(* CODESYS project boiler_olgovo_22_10_2019.project
   Company: syat
   Title: boiler_olgovo
   Author: User
   Version: 0.0.0.207

Project tree, tasks and I/O mapping:
  MyController : TM241CE40T/U, Schneider Electric, order no. TM241CE40T/U, version 4.0.6.18
      settings: OPCUA enable = False
    application Application
      libraries: CAA Real Time Clock Extern, 3.5.1.0 (CAA Technical Workgroup); SysTimeRtc, 3.5.1.0 (System)
      task MAST (cyclic, interval 20 ms, priority 15, watchdog 100 ms x 1) calls analog_input, IN_A1_A12_A14_A17, MB_IN, get_data_from_CKM, reset_flowmetr, send_data_to_flowmeter, zadanie_for_m1_m2, get_data_from_flowmetr, BURNERS_GAZ_GRU, avg, day_mode, HVO_HEATER, connection, DYMOHODS, RECIRCULATIONS_M5_M6_M7, POUWER_BOILER, ALL_ERR, zadanie_for_burner, set_time, ERR_SENSER, SECURITY_BOILER, VALVE_FEEDER_PUMP_FEEDERS_M3_M4, NET_PUMPS_M1_M2, TRHD_PEREPUSK, ZATVORS, MB_OUT, OUT_PIN, send_data_to_flowmeter
      global variables GVL
      program OUT_PIN [ST]
      program IN_A1_A12_A14_A17 [ST]
      FB/
        function block VALVE_FEEDER [LD]
        function block PUMP [LD]
        function block VALVE [LD]
        function block BURNER_SMALL [LD]
        function send_to_ckm [LD]
        function block VALVE_TRHD [LD]
        function block PUMP_PCH [LD]
        function block VALVE_DYMOHOD [LD]
        function block VALVE_TRHD_PEREPUSK [LD]
        function block BURNER_BIG [LD]
      program MB_OUT [ST]
      program MB_IN [ST]
      program DYMOHODS [LD]
      program ZATVORS [LD]
      program TRHD_PEREPUSK [LD]
      program HVO_HEATER [LD]
      program RECIRCULATIONS_M5_M6_M7 [LD]
      program NET_PUMPS_M1_M2 [LD]
      program VALVE_FEEDER_PUMP_FEEDERS_M3_M4 [LD]
      program SECURITY_BOILER [LD]
      program BURNERS_GAZ_GRU [LD]
      program POUWER_BOILER [ST]
      program get_data_from_flowmetr [ST]
      program get_data_from_CKM [ST]
      program get_data_from_gaz_korr [LD]
      program zadanie_for_burner [ST]
      program ERR_SENSER [LD]
      program ALL_ERR [LD]
      global variables GVL_RETAIN
      A_TESTS/
        program zadanie_for_m1_m2 [ST]
        program zadanie_for_pch_m7 [ST]
        program zadanie_m7 [FBD]
        program zadanie_m1_m2 [FBD]
      RecipeManager
      global variables GVL_state_valve
      global variables GVL_STATE_PUMP
      global variables GVL_grafik
      program send_data_to_flowmeter [LD]
      program reset_flowmetr [ST]
      program set_time [CFC]
      program day_mode [CFC]
      program analog_input [LD]
      program avg [CFC]
      program connection [LD]
    DI : Digital Inputs, Schneider Electric, version 4.0.6.18
        input  idwDI_IDW0 : DWORD  // IDW0
        input  X0 : BOOL  // IDW0.I0
        input  X1 : BOOL  // IDW0.I1
        input  X2 : BOOL  // IDW0.I2
        input  X3 : BOOL  // IDW0.I3
        input  X4 : BOOL  // IDW0.I4
        input  X5 : BOOL  // IDW0.I5
        input  X6 : BOOL  // IDW0.I6
        input  X7 : BOOL  // IDW0.I7
        input  X8 : BOOL  // IDW0.I8
        input  X9 : BOOL  // IDW0.I9
        input  X10 : BOOL  // IDW0.I10
        input  X11 : BOOL  // IDW0.I11
        input  X12 : BOOL  // IDW0.I12
        input  X13 : BOOL  // IDW0.I13
        input  X14 : BOOL  // IDW0.I14
        input  X15 : BOOL  // IDW0.I15
        input  X16 : BOOL  // IDW0.I16
        input  X17 : BOOL  // IDW0.I17
        input  X18 : BOOL  // IDW0.I18
        input  X19 : BOOL  // IDW0.I19
        input  X20 : BOOL  // IDW0.I20
        input  X21 : BOOL  // IDW0.I21
        input  X22 : BOOL  // IDW0.I22
        input  X23 : BOOL  // IDW0.I23
        input  ibDI_IB1 : BYTE  // IB1
    DQ : Digital Outputs, Schneider Electric, version 4.0.6.18
        output Y0 : BOOL  // QW0.Q0
        output Y1 : BOOL  // QW0.Q1
        output Y2 : BOOL  // QW0.Q2
        output Y3 : BOOL  // QW0.Q3
        output Y4 : BOOL  // QW0.Q4
        output Y5 : BOOL  // QW0.Q5
        output Y6 : BOOL  // QW0.Q6
        output Y7 : BOOL  // QW0.Q7
        output Y8 : BOOL  // QW0.Q8
        output Y9 : BOOL  // QW0.Q9
        output Y10 : BOOL  // QW0.Q10
        output Y11 : BOOL  // QW0.Q11
        output Y12 : BOOL  // QW0.Q12
        output Y13 : BOOL  // QW0.Q13
        output Y14 : BOOL  // QW0.Q14
        output Y15 : BOOL  // QW0.Q15
        output qbDQ_QB1 : BYTE  // QB1
        unmapped channels: QW0
    Counters : Counters, Schneider Electric, version 4.0.6.18
    Pulse_Generators : Pulse Generators, Schneider Electric, version 4.0.6.18
    Cartridge_1 : Cartridge, Schneider Electric, version 4.0.6.18
    Cartridge_2 : Cartridge, Schneider Electric, version 4.0.6.18
    IO_Bus : IO bus - TM3, Schneider Electric, version 4.0.6.18
      A1_7 : TM3TI4/G, Schneider Electric, order no. TM3TI4/G, version 1.0.1.5
          settings: KPI Configuration.KPI Configuration[0] = 35; KPI Configuration.KPI Configuration[1] = 35; KPI Configuration.KPI Configuration[2] = 35; KPI Configuration.KPI Configuration[3] = 35; KPI Configuration.KPI Configuration[5] = 0; KPI Configuration.KPI Configuration[7] = 0; KPI Configuration.KPI Configuration[9] = 0; KPI Configuration.KPI Configuration[11] = 0; KPI Configuration.KPI Configuration[12] = 32; KPI Configuration.KPI Configuration[13] = 78; KPI Configuration.KPI Configuration[14] = 32; KPI Configuration.KPI Configuration[15] = 78; KPI Configuration.KPI Configuration[16] = 32; KPI Configuration.KPI Configuration[17] = 78; KPI Configuration.KPI Configuration[18] = 32; KPI Configuration.KPI Configuration[19] = 78; KPI Configuration.KPI Configuration[20] = 10; KPI Configuration.KPI Configuration[22] = 10; KPI Configuration.KPI Configuration[24] = 10; KPI Configuration.KPI Configuration[26] = 10
          input  PT9 : INT  // IW0
          input  PT10 : INT  // IW1
          input  PT11 : INT  // IW2
          input  PT01 : INT  // IW3
          input  ERR_PT9 : BYTE  // IBStatusIW0
          input  ERR_PT10 : BYTE  // IBStatusIW1
          input  ERR_PT11 : BYTE  // IBStatusIW2
          input  ERR_PT01 : BYTE  // IBStatusIW3
      A1_6 : TM3AI8/G, Schneider Electric, order no. TM3AI8/G, version 1.0.0.17
          settings: KPI Configuration.KPI Configuration[0] = 35; KPI Configuration.KPI Configuration[1] = 35; KPI Configuration.KPI Configuration[2] = 35; KPI Configuration.KPI Configuration[3] = 35; KPI Configuration.KPI Configuration[4] = 35; KPI Configuration.KPI Configuration[5] = 35; KPI Configuration.KPI Configuration[6] = 35; KPI Configuration.KPI Configuration[7] = 35; KPI Configuration.KPI Configuration[9] = 0; KPI Configuration.KPI Configuration[11] = 0; KPI Configuration.KPI Configuration[13] = 0; KPI Configuration.KPI Configuration[15] = 0; KPI Configuration.KPI Configuration[17] = 0; KPI Configuration.KPI Configuration[19] = 0; KPI Configuration.KPI Configuration[21] = 0; KPI Configuration.KPI Configuration[23] = 0; KPI Configuration.KPI Configuration[24] = 32; KPI Configuration.KPI Configuration[25] = 78; KPI Configuration.KPI Configuration[26] = 32; KPI Configuration.KPI Configuration[27] = 78; KPI Configuration.KPI Configuration[28] = 32; KPI Configuration.KPI Configuration[29] = 78; KPI Configuration.KPI Configuration[30] = 32; KPI Configuration.KPI Configuration[31] = 78; KPI Configuration.KPI Configuration[32] = 32; KPI Configuration.KPI Configuration[33] = 78; KPI Configuration.KPI Configuration[34] = 32; KPI Configuration.KPI Configuration[35] = 78; KPI Configuration.KPI Configuration[36] = 32; KPI Configuration.KPI Configuration[37] = 78; KPI Configuration.KPI Configuration[38] = 32; KPI Configuration.KPI Configuration[39] = 78; KPI Configuration.KPI Configuration[40] = 10; KPI Configuration.KPI Configuration[42] = 10; KPI Configuration.KPI Configuration[44] = 10; KPI Configuration.KPI Configuration[46] = 10; KPI Configuration.KPI Configuration[48] = 10; KPI Configuration.KPI Configuration[50] = 10; KPI Configuration.KPI Configuration[52] = 10; KPI Configuration.KPI Configuration[54] = 10
          input  PT1 : INT  // IW0
          input  PT2 : INT  // IW1
          input  PT3 : INT  // IW2
          input  PT4 : INT  // IW3
          input  PT5 : INT  // IW4
          input  PT6 : INT  // IW5
          input  PT7 : INT  // IW6
          input  PT8 : INT  // IW7
          input  ERR_PT1 : BYTE  // IBStatusIW0
          input  ERR_PT2 : BYTE  // IBStatusIW1
          input  ERR_PT3 : BYTE  // IBStatusIW2
          input  ERR_PT4 : BYTE  // IBStatusIW3
          input  ERR_PT5 : BYTE  // IBStatusIW4
          input  ERR_PT6 : BYTE  // IBStatusIW5
          input  ERR_PT7 : BYTE  // IBStatusIW6
          input  ERR_PT8 : BYTE  // IBStatusIW7
      A1_5 : TM3AI8/G, Schneider Electric, order no. TM3AI8/G, version 1.0.0.17
          settings: KPI Configuration.KPI Configuration[0] = 35; KPI Configuration.KPI Configuration[1] = 35; KPI Configuration.KPI Configuration[2] = 35; KPI Configuration.KPI Configuration[3] = 35; KPI Configuration.KPI Configuration[4] = 35; KPI Configuration.KPI Configuration[5] = 35; KPI Configuration.KPI Configuration[6] = 35; KPI Configuration.KPI Configuration[7] = 35; KPI Configuration.KPI Configuration[9] = 0; KPI Configuration.KPI Configuration[11] = 0; KPI Configuration.KPI Configuration[13] = 0; KPI Configuration.KPI Configuration[15] = 0; KPI Configuration.KPI Configuration[17] = 0; KPI Configuration.KPI Configuration[19] = 0; KPI Configuration.KPI Configuration[21] = 0; KPI Configuration.KPI Configuration[23] = 0; KPI Configuration.KPI Configuration[24] = 32; KPI Configuration.KPI Configuration[25] = 78; KPI Configuration.KPI Configuration[26] = 32; KPI Configuration.KPI Configuration[27] = 78; KPI Configuration.KPI Configuration[28] = 32; KPI Configuration.KPI Configuration[29] = 78; KPI Configuration.KPI Configuration[30] = 32; KPI Configuration.KPI Configuration[31] = 78; KPI Configuration.KPI Configuration[32] = 32; KPI Configuration.KPI Configuration[33] = 78; KPI Configuration.KPI Configuration[34] = 208; KPI Configuration.KPI Configuration[35] = 7; KPI Configuration.KPI Configuration[36] = 32; KPI Configuration.KPI Configuration[37] = 78; KPI Configuration.KPI Configuration[38] = 32; KPI Configuration.KPI Configuration[39] = 78; KPI Configuration.KPI Configuration[40] = 10; KPI Configuration.KPI Configuration[42] = 10; KPI Configuration.KPI Configuration[44] = 10; KPI Configuration.KPI Configuration[46] = 10; KPI Configuration.KPI Configuration[48] = 10; KPI Configuration.KPI Configuration[50] = 10; KPI Configuration.KPI Configuration[52] = 10; KPI Configuration.KPI Configuration[54] = 10;
            KPI Configuration.KPI Configuration[61] = 1; KPI Configuration.KPI Configuration[62] = 1
          input  TT9 : INT  // IW0
          input  TT10 : INT  // IW1
          input  TT11 : INT  // IW2
          input  TT12 : INT  // IW3
          input  TT13 : INT  // IW4
          input  TT14 : INT  // IW5
          input  TT15 : INT  // IW6
          input  TT16 : INT  // IW7
          input  ERR_TT9 : BYTE  // IBStatusIW0
          input  ERR_TT10 : BYTE  // IBStatusIW1
          input  ERR_TT11 : BYTE  // IBStatusIW2
          input  ERR_TT12 : BYTE  // IBStatusIW3
          input  ERR_TT13 : BYTE  // IBStatusIW4
          input  ERR_TT14 : BYTE  // IBStatusIW5
          input  ERR_TT15 : BYTE  // IBStatusIW6
          input  ERR_TT16 : BYTE  // IBStatusIW7
      A1_4 : TM3AI8/G, Schneider Electric, order no. TM3AI8/G, version 1.0.0.17
          settings: KPI Configuration.KPI Configuration[0] = 35; KPI Configuration.KPI Configuration[1] = 35; KPI Configuration.KPI Configuration[2] = 35; KPI Configuration.KPI Configuration[3] = 35; KPI Configuration.KPI Configuration[4] = 35; KPI Configuration.KPI Configuration[5] = 35; KPI Configuration.KPI Configuration[6] = 35; KPI Configuration.KPI Configuration[7] = 35; KPI Configuration.KPI Configuration[9] = 0; KPI Configuration.KPI Configuration[11] = 0; KPI Configuration.KPI Configuration[13] = 0; KPI Configuration.KPI Configuration[15] = 0; KPI Configuration.KPI Configuration[17] = 0; KPI Configuration.KPI Configuration[19] = 0; KPI Configuration.KPI Configuration[21] = 0; KPI Configuration.KPI Configuration[23] = 0; KPI Configuration.KPI Configuration[24] = 32; KPI Configuration.KPI Configuration[25] = 78; KPI Configuration.KPI Configuration[26] = 32; KPI Configuration.KPI Configuration[27] = 78; KPI Configuration.KPI Configuration[28] = 32; KPI Configuration.KPI Configuration[29] = 78; KPI Configuration.KPI Configuration[30] = 32; KPI Configuration.KPI Configuration[31] = 78; KPI Configuration.KPI Configuration[32] = 32; KPI Configuration.KPI Configuration[33] = 78; KPI Configuration.KPI Configuration[34] = 32; KPI Configuration.KPI Configuration[35] = 78; KPI Configuration.KPI Configuration[36] = 32; KPI Configuration.KPI Configuration[37] = 78; KPI Configuration.KPI Configuration[38] = 32; KPI Configuration.KPI Configuration[39] = 78; KPI Configuration.KPI Configuration[40] = 10; KPI Configuration.KPI Configuration[42] = 10; KPI Configuration.KPI Configuration[44] = 10; KPI Configuration.KPI Configuration[46] = 10; KPI Configuration.KPI Configuration[48] = 10; KPI Configuration.KPI Configuration[50] = 10; KPI Configuration.KPI Configuration[52] = 10; KPI Configuration.KPI Configuration[54] = 10
          input  TT1 : INT  // IW0
          input  TT2 : INT  // IW1
          input  TT3 : INT  // IW2
          input  TT4 : INT  // IW3
          input  TT5 : INT  // IW4
          input  TT6 : INT  // IW5
          input  TT7 : INT  // IW6
          input  TT8 : INT  // IW7
          input  ERR_TT1 : BYTE  // IBStatusIW0
          input  ERR_TT2 : BYTE  // IBStatusIW1
          input  ERR_TT3 : BYTE  // IBStatusIW2
          input  ERR_TT4 : BYTE  // IBStatusIW3
          input  ERR_TT5 : BYTE  // IBStatusIW4
          input  ERR_TT6 : BYTE  // IBStatusIW5
          input  ERR_TT7 : BYTE  // IBStatusIW6
          input  ERR_TT8 : BYTE  // IBStatusIW7
      A1_3 : TM3DQ32TK, Schneider Electric, order no. TM3DQ32TK, version 1.0.1.3
          output IY0 : BOOL  // QD0.Q0
          output IY1 : BOOL  // QD0.Q1
          output IY2 : BOOL  // QD0.Q2
          output IY3 : BOOL  // QD0.Q3
          output IY4 : BOOL  // QD0.Q4
          output IY5 : BOOL  // QD0.Q5
          output IY6 : BOOL  // QD0.Q6
          output IY7 : BOOL  // QD0.Q7
          output IY8 : BOOL  // QD0.Q8
          output IY9 : BOOL  // QD0.Q9
          output IY10 : BOOL  // QD0.Q10
          output IY11 : BOOL  // QD0.Q11
          output IY12 : BOOL  // QD0.Q12
          output IY13 : BOOL  // QD0.Q13
          output IY14 : BOOL  // QD0.Q14
          output IY15 : BOOL  // QD0.Q15
          output IY16 : BOOL  // QD0.Q16
          output IY17 : BOOL  // QD0.Q17
          output IY18 : BOOL  // QD0.Q18
          output IY19 : BOOL  // QD0.Q19
          output IY20 : BOOL  // QD0.Q20
          output IY25 : BOOL  // QD0.Q25
          unmapped channels: QD0
      A1_1 : TM3DI32K, Schneider Electric, order no. TM3DI32K, version 1.0.1.3
          input  idwA1_1_ID0 : DWORD  // ID0
          input  IX0 : BOOL  // ID0.I0
          input  IX1 : BOOL  // ID0.I1
          input  IX2 : BOOL  // ID0.I2
          input  IX3 : BOOL  // ID0.I3
          input  IX4 : BOOL  // ID0.I4
          input  IX5 : BOOL  // ID0.I5
          input  IX6 : BOOL  // ID0.I6
          input  IX7 : BOOL  // ID0.I7
          input  IX8 : BOOL  // ID0.I8
          input  IX9 : BOOL  // ID0.I9
          input  IX10 : BOOL  // ID0.I10
          input  IX11 : BOOL  // ID0.I11
          input  IX12 : BOOL  // ID0.I12
          input  IX13 : BOOL  // ID0.I13
          input  IX14 : BOOL  // ID0.I14
          input  IX15 : BOOL  // ID0.I15
          input  IX16 : BOOL  // ID0.I16
          input  IX17 : BOOL  // ID0.I17
          input  IX18 : BOOL  // ID0.I18
          input  IX19 : BOOL  // ID0.I19
          input  IX20 : BOOL  // ID0.I20
          input  IX21 : BOOL  // ID0.I21
          input  IX22 : BOOL  // ID0.I22
          input  IX23 : BOOL  // ID0.I23
          input  IX24 : BOOL  // ID0.I24
          input  IX25 : BOOL  // ID0.I25
          input  IX26 : BOOL  // ID0.I26
          input  IX27 : BOOL  // ID0.I27
          input  IX28 : BOOL  // ID0.I28
          input  IX29 : BOOL  // ID0.I29
          input  IX30 : BOOL  // ID0.I30
          input  IX31 : BOOL  // ID0.I31
      A1_2 : TM3DI32K, Schneider Electric, order no. TM3DI32K, version 1.0.1.3
          input  IIX0 : BOOL  // ID0.I0
          input  IIX1 : BOOL  // ID0.I1
          input  IIX6 : BOOL  // ID0.I6
          input  IIX7 : BOOL  // ID0.I7
          input  IIX12 : BOOL  // ID0.I12
          input  IIX15 : BOOL  // ID0.I15
          unmapped channels: ID0
    COM_Bus : COM bus, Schneider Electric, version 4.0.6.18
    Ethernet_1 : Ethernet Network, Schneider Electric, version 4.0.6.18
        settings: IPAddress = [192, 168, 0, 32]; SubnetMask = [255, 255, 255, 0]; GatewayAddress = [192, 168, 0, 30]; DeviceName = 'plc_olgovo'; WebServer = TRUE; FTP Server = TRUE; SoMachine Protocol = TRUE; Modbus Server = TRUE; NetManage Protocol = TRUE; SNMP protocol = TRUE; Enable Routing = FALSE; WebVisu protocol = TRUE; DHCP Server Active = TRUE
    Serial_Line_1 : Serial line, Schneider Electric, version 4.0.6.18
      ASCII_Manager : ASCII Manager, Schneider Electric, version 4.0.0.2
    Serial_Line_2 : Serial line, Schneider Electric, version 4.0.6.18
      Modbus_IOScanner : Modbus IOScanner, Schneider Electric, version 3.5.3.8
          settings: Transmission = 'RTU'; ResponseTimeout = 1000; TimeBetweenFrames = 5
        Generic_Modbus_Slave : Generic Modbus Slave, Schneider Electric, version 3.5.3.9
            settings: SlaveAddress = 9; ResponseTimeout = 1000; Channel 1.Function Code = 4; Channel 1.Read Offset = 16#8000; Channel 1.Read Length = 2; Channel 1.Write Offset = 0; Channel 1.Write Length = 0; Channel 1.Cycle Time = 100; Channel 2.Function Code = 4; Channel 2.Read Offset = 16#C000; Channel 2.Read Length = 76; Channel 2.Write Offset = 0; Channel 2.Write Length = 0; Channel 2.Cycle Time = 100
            input  Application.skm_number_arr : ARRAY[0..1] OF WORD  // Channel 1
            input  Application.skm_all : ARRAY[0..75] OF WORD  // Channel 2
        OVEN : Generic Modbus Slave, Schneider Electric, version 3.5.3.9
            settings: SlaveAddress = 16; ResponseTimeout = 100; Channel 1.Function Code = 3; Channel 1.Read Offset = 16#0001; Channel 1.Read Length = 1; Channel 1.Write Offset = 0; Channel 1.Write Length = 0; Channel 1.Cycle Time = 100; Channel 2.Function Code = 3; Channel 2.Read Offset = 16#0007; Channel 2.Read Length = 1; Channel 2.Write Offset = 0; Channel 2.Write Length = 0; Channel 2.Cycle Time = 100
            input  Application.POSITION_VALVE_PEREPUSK : WORD  // Channel 1.Channel 1[0]
            input  Application.POSITION_VALVE_HEATER : WORD  // Channel 2.Channel 2[0]
            unmapped channels: Channel 1, Channel 2
        OVEN_OUT : Generic Modbus Slave, Schneider Electric, version 3.5.3.9
            settings: SlaveAddress = 17; ResponseTimeout = 101; Channel 1.Function Code = 16; Channel 1.Read Offset = 0; Channel 1.Read Length = 0; Channel 1.Write Offset = 16#0000; Channel 1.Write Length = 1; Channel 1.Cycle Time = 100; Channel 2.Function Code = 16; Channel 2.Read Offset = 0; Channel 2.Read Length = 0; Channel 2.Write Offset = 16#0001; Channel 2.Write Length = 1; Channel 2.Cycle Time = 100; Channel 3.Function Code = 16; Channel 3.Read Offset = 0; Channel 3.Read Length = 0; Channel 3.Write Offset = 16#0002; Channel 3.Write Length = 1; Channel 3.Cycle Time = 100
            output Application.PCH_PUMP_M1_ZADANIE : ARRAY[0..0] OF WORD  // Channel 1
            output Application.PCH_PUMP_M2_ZADANIE : ARRAY[0..0] OF WORD  // Channel 2
            output Application.PCH_PUMP_M7_ZADANIE : ARRAY[0..0] OF WORD  // Channel 3
        ek270a : Generic Modbus Slave, Schneider Electric, version 3.5.3.9
            settings: ek270.Function Code = 3; ek270.Read Offset = 16#0146; ek270.Read Length = 2; ek270.Write Offset = 0; ek270.Write Length = 0; ek270.Cycle Time = 100; Channel 2.Function Code = 3; Channel 2.Read Offset = 16#0148; Channel 2.Read Length = 2; Channel 2.Write Offset = 0; Channel 2.Write Length = 0; Channel 2.Cycle Time = 100; Channel 3.Function Code = 3; Channel 3.Read Offset = 16#0064; Channel 3.Read Length = 2; Channel 3.Write Offset = 0; Channel 3.Write Length = 0; Channel 3.Cycle Time = 100; Channel 4.Function Code = 3; Channel 4.Read Offset = 16#0066; Channel 4.Read Length = 2; Channel 4.Write Offset = 0; Channel 4.Write Length = 0; Channel 4.Cycle Time = 100
            input  Q_s : WORD  // ek270.ek270[0]
            input  Q_l : WORD  // ek270.ek270[1]
            input  Qb_s : WORD  // Channel 2.Channel 2[0]
            input  Qb_l : WORD  // Channel 2.Channel 2[1]
            input  V_s : WORD  // Channel 3.Channel 3[0]
            input  V_l : WORD  // Channel 3.Channel 3[1]
            input  Vb_s : WORD  // Channel 4.Channel 4[0]
            input  Vb_l : WORD  // Channel 4.Channel 4[1]
            unmapped channels: ek270, Channel 2, Channel 3, Channel 4
  FdtConnections : FDT Connections, Schneider Electric, version 1.0.0.2
  A_TESTS/
    program get_data_from_oven [ST]
    program zadanie_for_m1_m2 [ST]
    program zadanie_for_pch_m7 [ST]
    program zadanie_m7 [FBD]
    program zadanie_m1_m2 [FBD]
*)

// MyController/Application/GVL
VAR_GLOBAL
	
start_test : BOOL;

//БЛОК ДЛЯ ОБМЕНА С РАСХОДОМЕРОМ ======НАЧАЛО======	
  	FLOW_BOILER_1 AT %MD500: REAL;
	FLOW_BOILER_2 AT %MD501: REAL;
	fl_g_s AT %MW1004: WORD;
	fl_g_l AT %MW1006: WORD;
	FLOW_GAZ AT %MD502: DWORD;
	V_gaz AT %MD506:DWORD;
	//FLOW_BOILER И FL_BOILER ДОЛЖНЫ ССЫЛАТЬСЯ НА ОДНУ ПАМЯТЬ
	FL_BOILER_1 AT %MD500: DWORD;
	FL_BOILER_2 AT %MD501: DWORD;
	
	RASHOD_WATER AT %MW503: WORD;
	FL_HVO AT %MD504: DWORD;
	
//БЛОК ДЛЯ ОБМЕНА С РАСХОДОМЕРОМ ======КОЕЦ======
	
//БЛОК ДЛЯ ОБМЕНА С ОВЕНОМ ======НАЧАЛО======	
  	step: INT;
	POSITION_VALVE_PEREPUSK: INT;
	POSITION_VALVE_HEATER: INT; 
  	data_to_send: ARRAY[0..10] OF BYTE; 
  	resv_data_from_flowmtr_ADR6: ARRAY[0..10] OF BYTE;
	resv_data_from_flowmtr_ADR7: ARRAY[0..10] OF BYTE;
	resv_data_from_flowmtr_ADR8: ARRAY[0..10] OF BYTE;
	resv_data_from_ckm: ARRAY[0..120] OF BYTE;
	good: BOOL;
//БЛОК ДЛЯ ОБМЕНА С ОВЕНОМ ======КОЕЦ======

//БЛОК ОПИСАНИЯ ВХОДОВ А1_1  A1_2 =============НАЧАЛО=======
	ERR_PCH_PUMP_CYRCULATION AT %MX400.0: BOOL;
	ERR_PUMP1_CYRCULATION AT %MX400.1: BOOL;
	ERR_PUMP2_CYRCULATION AT %MX400.2: BOOL;
	ERR_PCH_PUMP1_NET AT %MX400.3: BOOL;
	ERR_PCH_PUMP2_NET AT %MX400.4: BOOL;
	ERR_M3_FEEDER AT %MX400.5: BOOL;
	ERR_M4_FEEDER AT %MX400.6: BOOL;
	VALVE_GAZ_OPENED AT %MX400.7: BOOL;
	VALVE_GAZ_CLOSED AT %MX400.8: BOOL;
	ERR_DEGAZATOR AT %MX400.9: BOOL;
	FIRE AT %MX400.10: BOOL;
	BREAKE AT %MX400.11: BOOL;
	N0_SECURITY AT %MX400.12: BOOL;
	SECURITY AT %MX400.13: BOOL;
	ERR_GAZ AT %MX400.14: BOOL;
	ERR_BURNER1 AT %MX400.15: BOOL;
	

	BTN_HAND_MODE_PUMPS: BOOL;
	BTN_AUTO_MODE_PUMPS:BOOL;
	BTN_HAND_MODE_BOILERS: BOOL;
	BTN_AUTO_MODE_BOILERS:BOOL;
	BTN_HAND_MODE_VALVES: BOOL;
	BTN_AUTO_MODE_VALVES:BOOL;
	BTN_START_BURNER: BOOL;
//БЛОК ОПИСАНИЯ ВХОДОВ А1_1 A1_2 =============КОНЕЦ========

//БЛОК ОПИСАНИЯ ВХОДОВ А1 =============НАЧАЛО=======
	ERR_BURNER2 AT %MX402.0: BOOL;
	BURNER2_WORKS AT %MX402.1: BOOL;
	DYMOHOD1_OPENED AT %MX402.2: BOOL;
	DYMOHOD1_CLOSED AT %MX402.3: BOOL;
	ZATVOR1_OPENED AT %MX402.4: BOOL;
	ZATVOR1_CLOSED AT %MX402.5: BOOL;
	DYMOHOD2_OPENED AT %MX402.6: BOOL;
	DYMOHOD2_CLOSED AT %MX402.7: BOOL;
	ZATVOR2_OPENED AT %MX402.8: BOOL;
	ZATVOR2_CLOSED AT %MX402.9: BOOL;
	FEEDER_OPENED AT %MX402.10: BOOL;
	FEEDER_CLOSED AT %MX402.11: BOOL;
	HVO_OPENED AT %MX402.12: BOOL;
	HVO_CLOSED AT %MX402.13: BOOL;
	PEREPUSK_OPENED AT %MX402.14: BOOL;
	PEREPUSK_CLOSED AT %MX402.15: BOOL;
		
//БЛОК ОПИСАНИЯ ВХОДОВ А1 =============КОНЕЦ========



//БЛОК ОПИСАНИЯ ВЫХОДОВ А1 =============НАЧАЛО=======
	HEATER_CLOSED AT %MX404.0: BOOL;
	OPEN_DYMOHOD1 AT %MX404.1: BOOL;
	CLOSE_DYMOHOD1 AT %MX404.2: BOOL;
	OPEN_ZATVOR1 AT %MX404.3: BOOL;
	CLOSE_ZATVOR1 AT %MX404.4: BOOL;
	OPEN_DYMOHOD2 AT %MX404.5: BOOL;
	CLOSE_DYMOHOD2 AT %MX404.6: BOOL;
	OPEN_ZATVOR2 AT %MX404.7: BOOL;
	CLOSE_ZATVOR2 AT %MX404.8: BOOL;
	OPEN_FEEDER AT %MX404.9: BOOL;
	CLOSE_FEEDER AT %MX404.10: BOOL;
	OPEN_HVO AT %MX404.11: BOOL;
	CLOSE_HVO AT %MX404.12: BOOL;
	OPEN_PEREPUSK AT %MX404.13: BOOL;
	CLOSE_PEREPUSK AT %MX404.14: BOOL;
	OPEN_HEATER AT %MX404.15: BOOL;

	CLOSE_HEATER AT %MX406.0: BOOL;
	BURNER1_WORKS AT %MX406.1: BOOL;	
	HEATER_OPENED AT %MX406.2: BOOL;
	
//БЛОК ОПИСАНИЯ ВЫХОДОВ А1 =============КОНЕЦ=======

//БЛОК ОПИСАНИЯ ВЫХОДОВ А1_1 =============НАЧАЛО=======
	RUN_PUMP_CYRCULATION AT %MX406.3: BOOL;
	RUN_PUMP_CYRCULATION1 AT %MX406.4: BOOL;
	RUN_PUMP_CYRCULATION2 AT %MX406.5: BOOL;
	RUN_PUMP1_NET AT %MX406.6: BOOL;
	RUN_PUMP2_NET AT %MX406.7: BOOL;
	RUN_M3_FEEDER AT %MX406.8: BOOL;
	RUN_M4_FEEDER AT %MX406.9: BOOL;
	OPEN_GAZ AT %MX406.10: BOOL;
	CLOSE_GAZ AT %MX406.11: BOOL;
	RUN_SIGNAL_FIRE AT %MX406.12: BOOL;
	RUN_SIGNAL_BREAKE AT %MX406.13: BOOL;
	RUN_SMALL_FIRE_BURNER1 AT %MX406.14: BOOL;
	RUN_LARGE_FIRE_BURNER1 AT %MX406.15: BOOL;
	
	RUN_SMALL_FIRE_BURNER2 AT %MX408.0: BOOL;
	RUN_LARGE_FIRE_BURNER2 AT %MX408.1: BOOL;
	RKF AT %MX408.11: BOOL;
	ERR_BURNER_1 AT %MX408.12: BOOL;
	ERR_BURNER_2 AT %MX408.13: BOOL;
	START_STOP_BURNER1: BOOL;
	START_STOP_BURNER2: BOOL;
	RUN_LIGHT_KOLONNA: BOOL;
	RUN_HAND_MODE_PUMPS: BOOL;
	RUN_HAND_MODE_BOILERS: BOOL;
	RUN_HAND_MODE_VALVES: BOOL;
//БЛОК ОПИСАНИЯ ВЫХОДОВ А1_1 =============КОНЕЦ=======

//БЛОК ОПИСАНИЯ АНАЛОГОЫХ ВХОДОВ А1_3==========НАЧАЛО======
	TT1_DYMA_1 AT %MW100: INT;
	TT2_WTR_IN_1 AT %MW101: INT;
	TT3_WTR_OUT_1 AT %MW102: INT;
	TT4_DYMA_UTIL_OUT AT %MW103: INT;
	TT5_DYMA_2 AT %MW104: INT;
	TT6_WTR_UTIL_IN AT %MW105: INT;
	TT7_WTR_IN_2 AT %MW106: INT;
	TT8_WTR_OUT_2 AT %MW107: INT;
	
	TT9_WTR_IN_3H AT %MW108: INT;
	TT10_WTR_OUT_3H AT %MW109: INT;
	TT11_NET_WTR_IN1 AT %MW110: INT;
	TT12_NET_WTR_OUT AT %MW111: INT;
	TT13_NET_WTR_IN2 AT %MW112: INT;
	TT14_WTR_FEDER AT %MW113: INT;
	TT15_IN_ROOM AT %MW114: INT;
	TT16_ON_AIR AT %MW115: INT;
	
	PT1_WTR_IN_1 AT %MW116: INT;
	PT2_WTR_OUT_1 AT %MW117: INT;
	PT3_WTR_UTIL_IN AT %MW118: INT;
	PT4_WTR_IN_2 AT %MW119: INT;
	PT5_WTR_OUT_2 AT %MW120: INT;
	PT6_WTR_IN_3H AT %MW121: INT;
	PT7_WTR_OUT_3H AT %MW122: INT;
	PT8_WTR_OUT_BOILER AT %MW123: INT;
	
	PT9_WTR_IN_BOILER AT %MW124: INT;
	PT10_LEVEL_HVO AT %MW125: INT;
	PT11_WTR_IN_BOILER AT %MW126: INT;
	PT01_GAZ AT %MW127: INT;
	
	MW128 AT %MW128: INT;//POSITION_VALVE_PEREPUSK
	MW129 AT %MW129: INT;//POSITION_VALVE_HEATER
	TT12_NET_WATER_ZADANIE AT %MW130:INT;//температура сетевой воды задание для трехходового переключателя потока
	
	//t1_recipes AT %MW132: INT;
	//t2_recipes AT %MW133: INT;

	PCH_PUMP_M1_ZADANIE: INT;
	PCH_PUMP_M2_ZADANIE: INT;
	PCH_PUMP_M7_ZADANIE: INT;
	FREQ_M1: INT;
	FREQ_M2: INT;
	FREQ_M7: INT;
	FREQUENCY_M1 AT %MW134: INT;
	FREQUENCY_M2 AT %MW135: INT;
	FREQUENCY_M7 AT %MW136: INT;
	
	
	
//БЛОК ОПИСАНИЯ АНАЛОГОЫХ ВХОДОВ А1_3 ========== КОНЕЦ ======

//БЛОК ОПИСАНИЯ ПЕРЕМЕННХ ДЛЯ ПЕРЕДАЧИ bool В ПАНЕЛЬ MB_OUT ========== НАЧАЛО ======
	
	//MW200 AT %MW200: WORD;
	//MW201 AT %MW201: WORD;
	//MW202 AT %MW202: WORD;
	//MW203 AT %MW203: WORD;
	//MW204 AT %MW204: WORD;
	//MW205 AT %MW205: WORD;
	//MW206 AT %MW206: WORD;
	MW207 AT %MW207: WORD;
	MW208 AT %MW208: WORD;
	//MW209 AT %MW209: WORD;
	//MW210 AT %MW210: WORD;
	//MW211 AT %MW211: WORD;
	//MW212 AT %MW212: WORD;
	
//БЛОК ОПИСАНИЯ ПЕРЕМЕННХ ДЛЯ ПЕРЕДАЧИ bool В ПАНЕЛЬ MB_OUT ========== КОНЕЦ ======

//БЛОК ОПИСАНИЯ ПЕРЕМЕННХ ГОРЕЛКИ ========== НАЧАЛО ======

	FLOW_WATER_1 AT %MW315: INT;
	FLOW_WATER_2 AT %MW316: INT;
	ERR_WIRING_TT3 : BOOL;
	ERR_WIRING_TT8: BOOL;
	ERR_WIRING: BOOL;
	USE_2_BOILERS: BOOL;
	
	POWER_BOILER_1: REAL; // РАСЧЕТНАЯ МОЩНОСТЬ КОТЛА 1
	POWER_BOILER_2: REAL; // РАСЧЕТНАЯ МОЩНОСТЬ КОТЛА 2
	POWER_GRAFIC: REAL; // ТРЕБУЕМАЯ МОЩНОСТЬ КОТЕЛНОЙ, РАСЧИТЫВАЕТСЯ ИСХОДЯ ИЗ ГРАФИКА ПОДАЧИ ВОДЫ

	
	T1_GRAFIC AT %MW317: INT;
	T2_GRAFIC AT %MW318: INT;
	
	ZADANIE_TMP_BURNER_1 AT %MW138: INT;
	ZADANIE_TMP_BURNER_2 AT %MW132: INT;

	
	
//БЛОК ОПИСАНИЯ ПЕРЕМЕННХ ГОРЕЛКИ ========== КОНЕЦ ======	

	START_BURNER1_MANUAL AT %MX408.2: BOOL;
	TBTN_ON_LAGE_FLAME_BURNER_1 AT %MX408.3: BOOL;
	START_BURNER2_MANUAL AT %MX408.4: BOOL;
	TBTN_ON_LAGE_FLAME_BURNER_2 AT %MX408.5: BOOL;
	HVO_EMPTY AT %MX408.6: BOOL;
	
//БИТЫ ВКЛЮЧЕНИЯ ВЫКЛЮЧЕНИЯ МЕХАНИЗМОВ ========== НАЧАЛО ======
	BTN_OPEN_DYMOHOD1 AT %MX410.0: BOOL;
	BTN_CLOSE_DYMOHOD1 AT %MX410.1: BOOL;
	BTN_OPEN_ZATVOR1 AT %MX410.2: BOOL;
	BTN_CLOSE_ZATVOR1 AT %MX410.3: BOOL;
	BTN_OPEN_DYMOHOD2 AT %MX410.4: BOOL;
	BTN_CLOSE_DYMOHOD2 AT %MX410.5: BOOL;
	BTN_OPEN_ZATVOR2 AT %MX410.6: BOOL;
	BTN_CLOSE_ZATVOR2 AT %MX410.7: BOOL;
	BTN_OPEN_FEEDER AT %MX410.8: BOOL;
	BTN_CLOSE_FEEDER AT %MX410.9: BOOL;
	BTN_OPEN_HVO AT %MX410.10: BOOL;
	BTN_CLOSE_HVO AT %MX410.11: BOOL;
	BTN_OPEN_PEREPUSK AT %MX410.12: BOOL;
	BTN_CLOSE_PEREPUSK AT %MX410.13: BOOL;
	BTN_OPEN_HEATER AT %MX410.14: BOOL;
	BTN_CLOSE_HEATER AT %MX410.15: BOOL;
	
	BTN_RUN_PUMP_CYRCULATION AT %MX412.0: BOOL;
	BTN_RUN_PUMP_CYRCULATION1 AT %MX412.1: BOOL;
	BTN_RUN_PUMP_CYRCULATION2 AT %MX412.2: BOOL;
	BTN_RUN_PUMP1_NET AT %MX412.3: BOOL;
	BTN_RUN_PUMP2_NET AT %MX412.4: BOOL;
	BTN_RUN_M3_FEEDER AT %MX412.5: BOOL;
	BTN_RUN_M4_FEEDER AT %MX412.6: BOOL;
	BTN_OPEN_GAZ AT %MX412.7: BOOL;
	BTN_CLOSE_GAZ AT %MX412.8: BOOL;
	BTN_RUN_SIGNAL_FIRE AT %MX412.9: BOOL;
	BTN_RUN_SIGNAL_BREAKE AT %MX412.10: BOOL;
	RESET_ERR AT %MX412.11: BOOL;
	
	AUTO_MODE AT %MX412.15: BOOL;
	
	//BTN_PUSK_STOP_BOILER: BOOL;
//БИТЫ ВКЛЮЧЕНИЯ ВЫКЛЮЧЕНИЯ МЕХАНИЗМОВ ========== КОНЕЦ ======	

	//AUTO_MODE: BOOL;
	//: BOOL;
	LEVEL_BAK_ZAPASA: BOOL;

	
	RASHOL_WATER: INT;
	ERR_SL_1: BOOL;
	ZADANIE: INT;
	MEDIUM_TEMP_AIR: INT;
	ERR_FLOW_IN_NET: BOOL;
	

	DYMOHOD_BURNER1: VALVE_DYMOHOD;
	DYMOHOD_BURNER2: VALVE_DYMOHOD;
	ZATVOR_BURNER1: VALVE;
	ZATVOR_BURNER2: VALVE;
	FEEDER_PB: VALVE_FEEDER;
	HEATER_BOILER: VALVE_TRHD;
	GAZ_GRU: VALVE;
	HVO_1: VALVE;
	PEREPUSK: VALVE_TRHD_PEREPUSK;
	PUMP_M7: PUMP_PCH;
	PUMP_M5: PUMP;
	PUMP_M6: PUMP;
	PUMP_M1: PUMP_PCH;
	PUMP_M2: PUMP_PCH;
	FEEDER_M3: PUMP;
	FEEDER_M4: PUMP;
	BURNER_1: BURNER_SMALL;
	BURNER_2: BURNER_BIG;
	send_data_to_flowmetr: SEND_RECV_MSG;
	ERR_PRES_GAZ: BOOL;
	ERR_POSITION_PEREPUSK: BOOL;
	
	ERR_SEN_TT1 AT %MX418.0: BOOL;
	ERR_SEN_TT2 AT %MX418.1: BOOL;
	ERR_SEN_TT3 AT %MX418.2: BOOL;
	ERR_SEN_TT4 AT %MX418.3: BOOL;
	ERR_SEN_TT5 AT %MX418.4: BOOL;
	ERR_SEN_TT6 AT %MX418.5: BOOL;
	ERR_SEN_TT7 AT %MX418.6: BOOL;
	ERR_SEN_TT8 AT %MX418.7: BOOL;
	ERR_SEN_TT9 AT %MX418.8: BOOL;
	ERR_SEN_TT10 AT %MX418.9: BOOL;
	ERR_SEN_TT11 AT %MX418.10: BOOL;
	ERR_SEN_TT12 AT %MX418.11: BOOL;
	ERR_SEN_TT13 AT %MX418.12: BOOL;
	ERR_SEN_TT14 AT %MX418.13: BOOL;
	ERR_SEN_TT15 AT %MX418.14: BOOL;
	ERR_SEN_TT16 AT %MX418.15: BOOL;
	
	ERR_SEN_PT1 AT %MX420.0: BOOL;
	ERR_SEN_PT2 AT %MX420.1: BOOL;
	ERR_SEN_PT3 AT %MX420.2: BOOL;
	ERR_SEN_PT4 AT %MX420.3: BOOL;
	ERR_SEN_PT5 AT %MX420.4: BOOL;
	ERR_SEN_PT6 AT %MX420.5: BOOL;
	ERR_SEN_PT7 AT %MX420.6: BOOL;
	ERR_SEN_PT8 AT %MX420.7: BOOL;
	ERR_SEN_PT9 AT %MX420.8: BOOL;
	ERR_SEN_PT10 AT %MX420.9: BOOL;
	ERR_SEN_PT11 AT %MX420.10: BOOL;
	ERR_SEN_PT01 AT %MX420.11: BOOL;
	ERR_TRMST_BURNER AT %MX420.12: BOOL;
	DA_ALL AT %MX420.13: BOOL;
	ERR_GERM_BURNER1 AT %MX420.14: BOOL;
	BURNER1_IN_AUTO_MODE AT %MX420.15: BOOL;
	
	ERR_GERM_BURNER2 AT %MX422.5: BOOL;
	BURNER2_IN_AUTO_MODE AT %MX422.6: BOOL;
	SMALL_PRESS AT %MX422.7: BOOL;
	delay_flame_visualisation1 AT  %MX422.9: BOOL;
	delay_flame_visualisation2 AT  %MX422.10: BOOL;

	BTN_PUSK_STOP_BOILER AT %MX422.3: BOOL;
	skm_number AT %MD600: UDINT;
	skm_number_arr : ARRAY[0..1] OF WORD;
	skm_all : ARRAY[0..75] OF WORD;
	skm_all_mw AT %MW1400: ARRAY[0..75] OF WORD;

	number_devise_l: INT; 
	number_devise_h: INT;
	number_devise_h1: INT;
	
	ERR_SEND_RECV_MSG: BOOL;
	

	off_light_kolonna AT %MX408.15: BOOL;
	RUN_DYMOHOD1_TO_OPEN: BOOL;
	RUN_DYMOHOD2_TO_OPEN: BOOL;
	ZADANIE_BALANSE_AVG: INT;
	
	connect_on AT %MX426.0: BOOL;
	connect_err AT %MX426.1: BOOL;
	
	event_cntr AT %MW986: INT;//Записать на флешку 
	
	ERR_PRESS_BOILER1 AT %MX426.2: BOOL;
	ERR_PRESS_BOILER2 AT %MX426.3: BOOL;
	ERR_GERM_BUR1: BOOL;
END_VAR;

// MyController/Application/GVL_RETAIN
VAR_GLOBAL RETAIN
	
	T_graf_1 AT %MW0: ARRAY[0..34] OF INT;
	T_graf_2 AT %MW40: ARRAY[0..34] OF INT;	
	
	
	TT15_IN_ROOM_ZADANIE AT %MW131: INT;//температура в комнате задание	
	
	Kp_m1 AT %MW140: INT;
	Tn_m1 AT %MW141: INT;
	Tv_m1 AT %MW142: INT;
	
	Kp_m7 AT %MW143: INT;
	Tn_m7 AT %MW144: INT;
	Tv_m7 AT %MW145: INT;

	Kp_m2 AT %MW146: INT;
	Tn_m2 AT %MW147: INT;
	Tv_m2 AT %MW148: INT;	
	
	TM_STOP AT %MW313: INT;
	PAUSE AT %MW314: INT;
	
	
	MANUAL_ZADANIE_TMP_BURNER1 AT %MW137: INT;//Ручное задание на выходе котла1	
	MANUAL_ZADANIE_TMP_BURNER2 AT %MW981: INT;//Ручное задание на выходе котла2	
	
	T_ZADANNOE AT %MW319: INT;
	MANUAL_ZADANIE_FOR_PCH AT %MW320: INT;// Задание для М1
	MANUAL_ZADANIE_FOR_PCH2 AT %MW325: INT;// Задание для М2
	
	MANUAL_ZADANIE_FOR_PCH_M7 AT %MW321: INT;
	
	PT8_WTR_OUT_BOILER_ZADANIE AT %MW322: INT;//ручное задание давления на подаче
	
	DELAY_CLOSE_ZATVOR_2 AT %MW323: INT;// Время закрытия дымохода 2
	DELAY_CLOSE_ZATVOR_1 AT %MW324: INT;
	
	PRIOR_BOILER_1 AT %MX412.12: BOOL;
	PRIOR_BOILER_2 AT %MX412.13: BOOL;
	PRIOR_PUMP_M5 AT %MX412.14: BOOL;
	
	PRIOR_PUMP_M6 AT %MX422.0: BOOL;
	PRIOR_PUMP_M1 AT %MX422.1: BOOL;
	PRIOR_PUMP_M2 AT %MX422.2: BOOL;
	PRIOR_PUMP_M3 AT %MX408.7: BOOL;
	PRIOR_PUMP_M4 AT %MX408.8: BOOL;
	err_floy_boiler_1 AT %MX408.9: BOOL;
	err_floy_boiler_2 AT %MX408.10: BOOL;
	
	xCommandSetRtc AT %MX408.14: BOOL;
	
	recirculation_M6_AUTO AT %MX422.4: BOOL;
	use_balanse_power AT %MX422.8: BOOL;
	
	DYMOHOD2_AUTO AT %MX424.0: BOOL;
	DYMOHOD1_AUTO AT %MX424.1: BOOL;
	ZATVOR1_AUTO AT %MX424.2: BOOL; 
	ZATVOR2_AUTO AT %MX424.3: BOOL;
	HVO_AUTO AT %MX424.4: BOOL;
	FEEDER_AUTO AT %MX424.5: BOOL;
	HEATER_AUTO AT %MX424.6: BOOL;
	PEREPUSK_AUTO AT %MX424.7: BOOL;
	BURNER1_AUTO AT %MX424.8: BOOL;
	BURNER2_AUTO AT %MX424.9: BOOL;
	RECIRCULATION_M7_AUTO AT %MX424.10: BOOL;
	PUMP_NET_M1_AUTO AT %MX424.11: BOOL;
	PUMP_NET_M2_AUTO AT %MX424.12: BOOL;
	FEEDER_M3_AUTO AT %MX424.13: BOOL;
	FEEDER_M4_AUTO AT %MX424.14: BOOL;
	recirculation_M5_AUTO AT %MX424.15: BOOL;
	
	
	DELTA_P_IN_OUT AT %MW800: INT;	
	min_P_gaz AT %MW801: INT;
	Kp_perepusk AT %MW802: INT;
	TN_perepusk AT %MW803: INT;
	TV_perepusk AT %MW804: INT;
	Kp_heater AT %MW805: INT;
	TN_heater AT %MW806: INT;
	TV_heater AT %MW807: INT;
	level_hvo_min AT %MW808: INT;
	level_hvo_max AT %MW809: INT;
	PT9_WTR_IN_BOILER_ZADANIE AT %MW810: INT;
	tmp_run_small_flame AT %MW811: INT;
	tmp_off_burner AT %MW812: INT;
	tmp_run_small_flame2 AT %MW813: INT;
	tmp_off_burner2 AT %MW814: INT;	
	min_rashod_boiler_1 AT %MW815: INT;
	min_rashod_boiler_2 AT %MW816: INT;
	tmp_use_1_and_2_boiler AT %MW817: INT;
	
	  uiSetYear AT %MW900: UINT; 
      uiSetMonth AT %MW901: UINT; 
      uiSetDay AT %MW902: UINT; 
      uiSetHour AT %MW903: UINT; 
      uiSetMinute AT %MW904: UINT; 
      uiSetSecond AT %MW905: UINT; 
      uiSetMSecond AT %MW906: UINT;
	  
	  DayModeHourStart AT %MW907: UINT;
	  DayModeMinuteStart AT %MW908: UINT;
	  DayModeHourStop AT %MW909: UINT;
	  DayModeMinuteStop AT %MW910: UINT;
	  DayModeTempAir AT %MW911: INT;
	  DayModeTempWater AT %MW912: INT;
	  ManZadaniePerepusk AT %MW913: INT;
	  MinPerepusk AT %MW914: INT;
	  MaxPerepusk AT %MW915: INT;
	  
	  t1Min AT %MW916: INT;
	  t1Max AT %MW917: INT;
	  
	  t2Min AT %MW918: INT;
	  t2Max AT %MW919: INT;
	  
	  t3Min AT %MW920: INT;
	  t3Max AT %MW921: INT;
	  
	  t4Min AT %MW922: INT;
	  t4Max AT %MW923: INT;
	  
	  t5Min AT %MW924: INT;
	  t5Max AT %MW925: INT;
	  	  
	  t6Min AT %MW926: INT;
	  t6Max AT %MW927: INT;
	  	  
	  t7Min AT %MW928: INT;
	  t7Max AT %MW929: INT;
	  	  
	  t8Min AT %MW930: INT;
	  t8Max AT %MW931: INT;
	  
	  t9Min AT %MW932: INT;
	  t9Max AT %MW933: INT;
	  
	  t10Min AT %MW934: INT;
	  t10Max AT %MW935: INT;
	  
	  t11Min AT %MW936: INT;
	  t11Max AT %MW937: INT;
	  
	  t12Min AT %MW938: INT;
	  t12Max AT %MW939: INT;
	  
	  t13Min AT %MW940: INT;
	  t13Max AT %MW941: INT;
	  	  
	  t14Min AT %MW942: INT;
	  t14Max AT %MW943: INT;
	  	  
	  t15Min AT %MW944: INT;
	  t15Max AT %MW945: INT;
	  	  
	  t16Min AT %MW946: INT;
	  t16Max AT %MW947: INT; 
	  	  
	  p1Min AT %MW948: INT;
	  p1Max AT %MW949: INT; 
	  	  
	  p2Min AT %MW950: INT;
	  p2Max AT %MW951: INT;
 	  	  
	  p3Min AT %MW952: INT;
	  p3Max AT %MW953: INT;    
 	  	  
	  p4Min AT %MW954: INT;
	  p4Max AT %MW955: INT;
 	  	  
	  p5Min AT %MW956: INT;
	  p5Max AT %MW957: INT; 
 	  	  
	  p6Min AT %MW958: INT;
	  p6Max AT %MW959: INT; 
 	  	  
	  p7Min AT %MW960: INT;
	  p7Max AT %MW961: INT;
 	  	  
	  p8Min AT %MW962: INT;
	  p8Max AT %MW963: INT; 
 	  	  
	  p9Min AT %MW964: INT;
	  p9Max AT %MW965: INT;
 	  	  
	  p10Min AT %MW966: INT;
	  p10Max AT %MW967: INT; 
 	  	  
	  p11Min AT %MW968: INT;
	  p11Max AT %MW969: INT;
 	  	  
	  p01Min AT %MW970: INT;
	  p01Max AT %MW971: INT;
	  
	  FLOW_GRAFIC AT %MW972: INT;
	  K AT %MW973: INT;
	  Tf AT %MW974: INT;
	  
	  TMP_OBRATKA AT %MW975: INT;
	  TMP_PODACHA AT %MW976: INT;
	  ZADANIE_BALANSE AT %MW977: INT;
	  MAX_TEMP_BALANSE AT %MW978: INT;
	  power_boiler1 AT %MW979: INT;//ЗАДАННАЯ МОЩНОСТЬ КОТЛА 1 С ПАНЕЛИ
	  power_boiler2 AT %MW980: INT;//ЗАДАННАЯ МОЩНОСТЬ КОТЛА 2 С ПАНЕЛИ
	  power_utilizator AT %MD491: REAL;
	  
	  //event_cntr AT %MW986: INT;
	  	
END_VAR

// MyController/Application/GVL_state_valve
VAR_GLOBAL
	GAZ_GRU_STATE AT %MW400: INT;
	DYMOHOD_BURNER1_STATE AT %MW401: INT;
	DYMOHOD_BURNER2_STATE AT %MW402: INT;
	HVO_STATE AT %MW403: INT;
	HEATER_BOILER_STATE AT %MW404: INT;
	PEREPUSK_STATE AT %MW405: INT;
	FEEDER_PB_STATE AT %MW406: INT;
	ZATVOR_BURNER1_STATE AT %MW407: INT;
	ZATVOR_BURNER2_STATE AT %MW408: INT;
END_VAR

// MyController/Application/GVL_STATE_PUMP
VAR_GLOBAL
	PUMP_M1_STATE AT %MW409: INT;
	PUMP_M2_STATE AT %MW410: INT;
	FEEDER_M3_STATE AT %MW411: INT;
	FEEDER_M4_STATE AT %MW412: INT;
	PUMP_M5_STATE AT %MW413: INT;
	PUMP_M6_STATE AT %MW414: INT;
	PUMP_M7_STATE AT %MW415: INT;	
END_VAR

// MyController/Application/GVL_grafik
VAR_GLOBAL
END_VAR

// MyController/Application/analog_input
PROGRAM analog_input
VAR
	sTT1: LIN_TRAFO;
	sTT2: LIN_TRAFO;
	sTT3: LIN_TRAFO;
	sTT4: LIN_TRAFO;
	sTT5: LIN_TRAFO;
	sTT6: LIN_TRAFO;
	sTT7: LIN_TRAFO;
	sTT8: LIN_TRAFO;
	sTT16: LIN_TRAFO;
	sTT15: LIN_TRAFO;
	sTT14: LIN_TRAFO;
	sTT13: LIN_TRAFO;
	sTT12: LIN_TRAFO;
	sTT11: LIN_TRAFO;
	sTT10: LIN_TRAFO;
	sTT9: LIN_TRAFO;
	sPT1: LIN_TRAFO;
	sPT2: LIN_TRAFO;
	sPT3: LIN_TRAFO;
	sPT4: LIN_TRAFO;
	sPT5: LIN_TRAFO;
	sPT6: LIN_TRAFO;
	sPT7: LIN_TRAFO;
	sPT8: LIN_TRAFO;
	sPT9: LIN_TRAFO;
	sPT10: LIN_TRAFO;
	sPT11: LIN_TRAFO;
	sPT01: LIN_TRAFO;
END_VAR

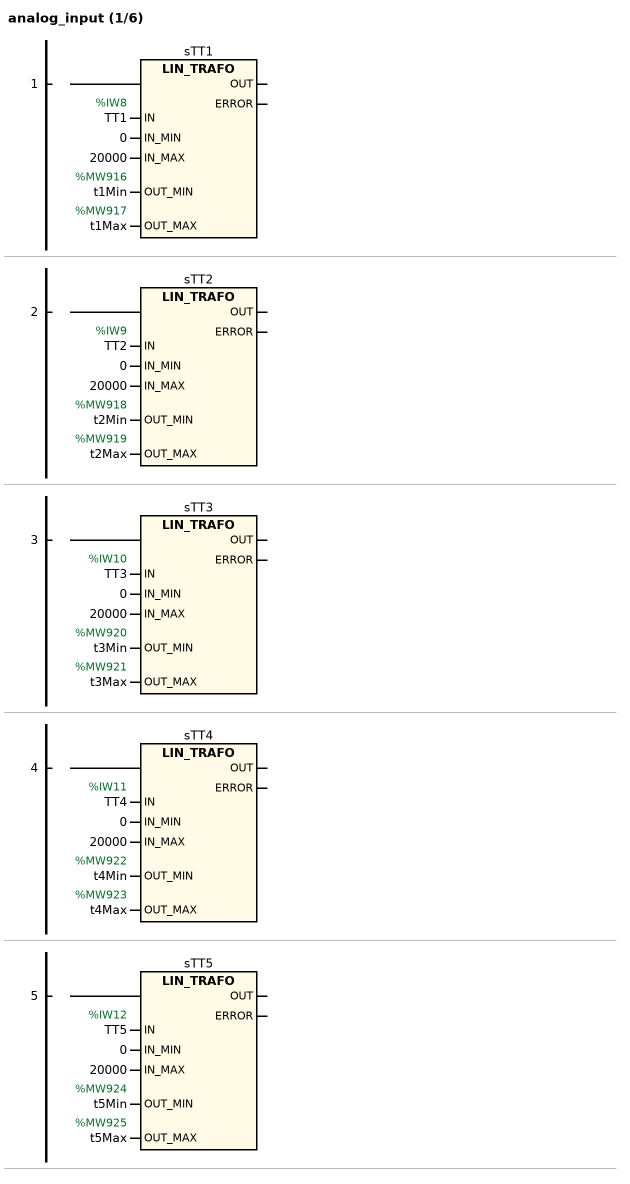
// NETWORK 1
//   TT1: A1_4 : | AT %IW8
//   t1Min: AT %MW916
//   t1Max: AT %MW917
sTT1(IN := TT1, IN_MIN := 0, IN_MAX := 20000, OUT_MIN := t1Min, OUT_MAX := t1Max); // LIN_TRAFO

// NETWORK 2
//   TT2: A1_4 : | AT %IW9
//   t2Min: AT %MW918
//   t2Max: AT %MW919
sTT2(IN := TT2, IN_MIN := 0, IN_MAX := 20000, OUT_MIN := t2Min, OUT_MAX := t2Max); // LIN_TRAFO

// NETWORK 3
//   TT3: A1_4 : | AT %IW10
//   t3Min: AT %MW920
//   t3Max: AT %MW921
sTT3(IN := TT3, IN_MIN := 0, IN_MAX := 20000, OUT_MIN := t3Min, OUT_MAX := t3Max); // LIN_TRAFO

// NETWORK 4
//   TT4: A1_4 : | AT %IW11
//   t4Min: AT %MW922
//   t4Max: AT %MW923
sTT4(IN := TT4, IN_MIN := 0, IN_MAX := 20000, OUT_MIN := t4Min, OUT_MAX := t4Max); // LIN_TRAFO

// NETWORK 5
//   TT5: A1_4 : | AT %IW12
//   t5Min: AT %MW924
//   t5Max: AT %MW925
sTT5(IN := TT5, IN_MIN := 0, IN_MAX := 20000, OUT_MIN := t5Min, OUT_MAX := t5Max); // LIN_TRAFO

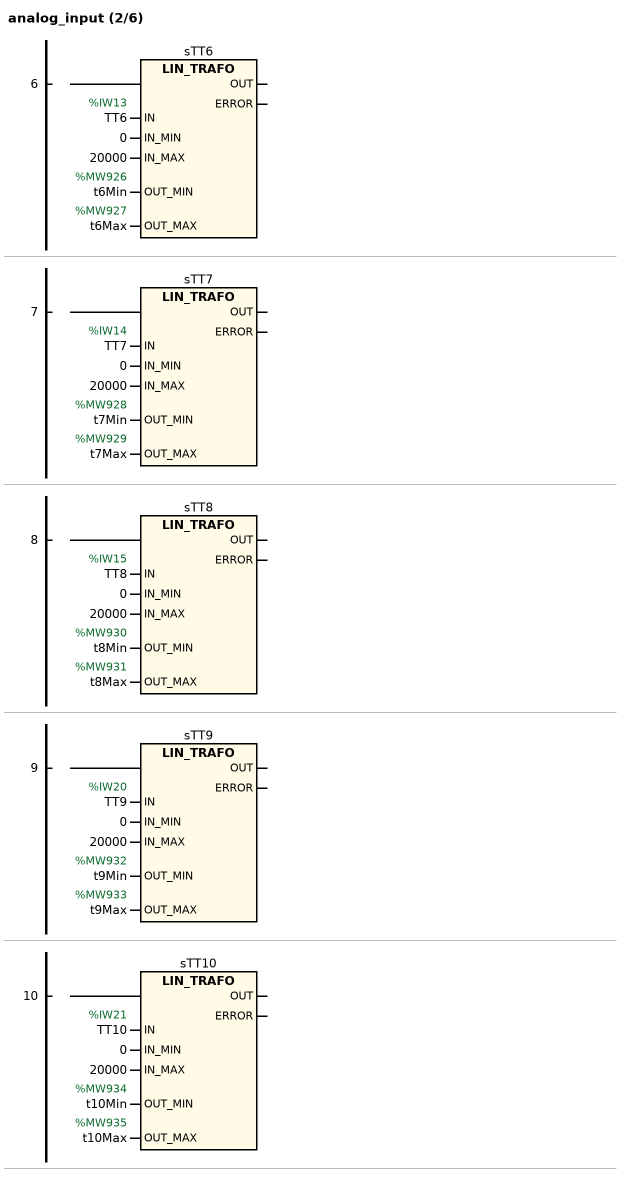
// NETWORK 6
//   TT6: A1_4 : | AT %IW13
//   t6Min: AT %MW926
//   t6Max: AT %MW927
sTT6(IN := TT6, IN_MIN := 0, IN_MAX := 20000, OUT_MIN := t6Min, OUT_MAX := t6Max); // LIN_TRAFO

// NETWORK 7
//   TT7: A1_4 : | AT %IW14
//   t7Min: AT %MW928
//   t7Max: AT %MW929
sTT7(IN := TT7, IN_MIN := 0, IN_MAX := 20000, OUT_MIN := t7Min, OUT_MAX := t7Max); // LIN_TRAFO

// NETWORK 8
//   TT8: A1_4 : | AT %IW15
//   t8Min: AT %MW930
//   t8Max: AT %MW931
sTT8(IN := TT8, IN_MIN := 0, IN_MAX := 20000, OUT_MIN := t8Min, OUT_MAX := t8Max); // LIN_TRAFO

// NETWORK 9
//   TT9: A1_5 : | AT %IW20
//   t9Min: AT %MW932
//   t9Max: AT %MW933
sTT9(IN := TT9, IN_MIN := 0, IN_MAX := 20000, OUT_MIN := t9Min, OUT_MAX := t9Max); // LIN_TRAFO

// NETWORK 10
//   TT10: A1_5 : | AT %IW21
//   t10Min: AT %MW934
//   t10Max: AT %MW935
sTT10(IN := TT10, IN_MIN := 0, IN_MAX := 20000, OUT_MIN := t10Min, OUT_MAX := t10Max); // LIN_TRAFO

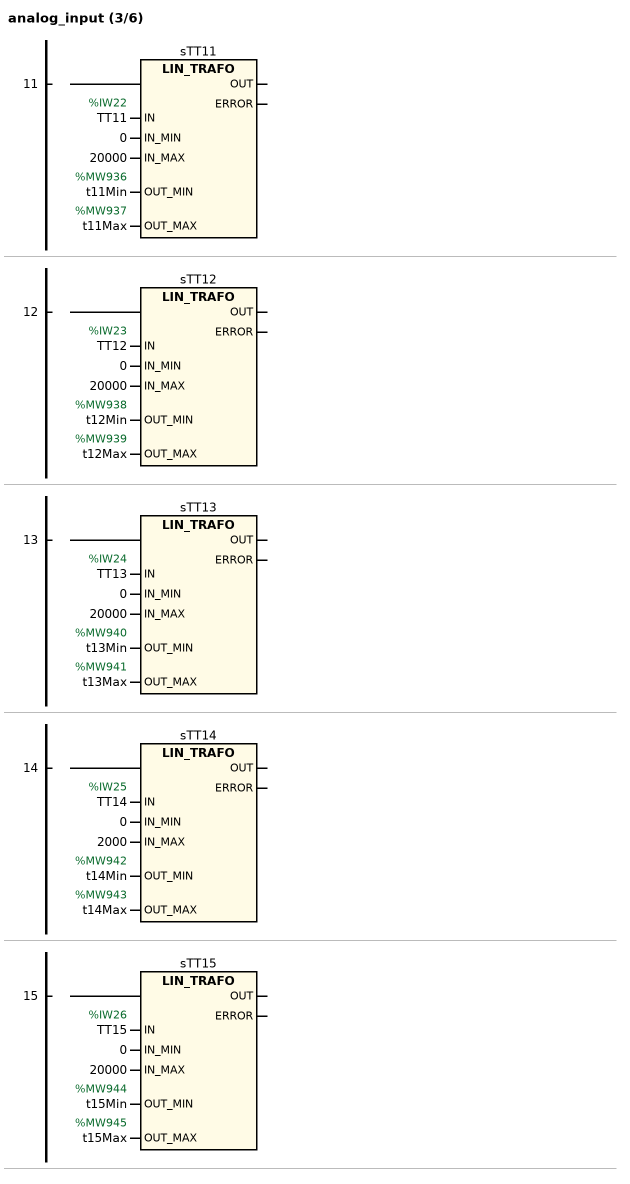
// NETWORK 11
//   TT11: A1_5 : | AT %IW22
//   t11Min: AT %MW936
//   t11Max: AT %MW937
sTT11(IN := TT11, IN_MIN := 0, IN_MAX := 20000, OUT_MIN := t11Min, OUT_MAX := t11Max); // LIN_TRAFO

// NETWORK 12
//   TT12: A1_5 : | AT %IW23
//   t12Min: AT %MW938
//   t12Max: AT %MW939
sTT12(IN := TT12, IN_MIN := 0, IN_MAX := 20000, OUT_MIN := t12Min, OUT_MAX := t12Max); // LIN_TRAFO

// NETWORK 13
//   TT13: A1_5 : | AT %IW24
//   t13Min: AT %MW940
//   t13Max: AT %MW941
sTT13(IN := TT13, IN_MIN := 0, IN_MAX := 20000, OUT_MIN := t13Min, OUT_MAX := t13Max); // LIN_TRAFO

// NETWORK 14
//   TT14: A1_5 : | AT %IW25
//   t14Min: AT %MW942
//   t14Max: AT %MW943
sTT14(IN := TT14, IN_MIN := 0, IN_MAX := 2000, OUT_MIN := t14Min, OUT_MAX := t14Max); // LIN_TRAFO

// NETWORK 15
//   TT15: A1_5 : | AT %IW26
//   t15Min: AT %MW944
//   t15Max: AT %MW945
sTT15(IN := TT15, IN_MIN := 0, IN_MAX := 20000, OUT_MIN := t15Min, OUT_MAX := t15Max); // LIN_TRAFO

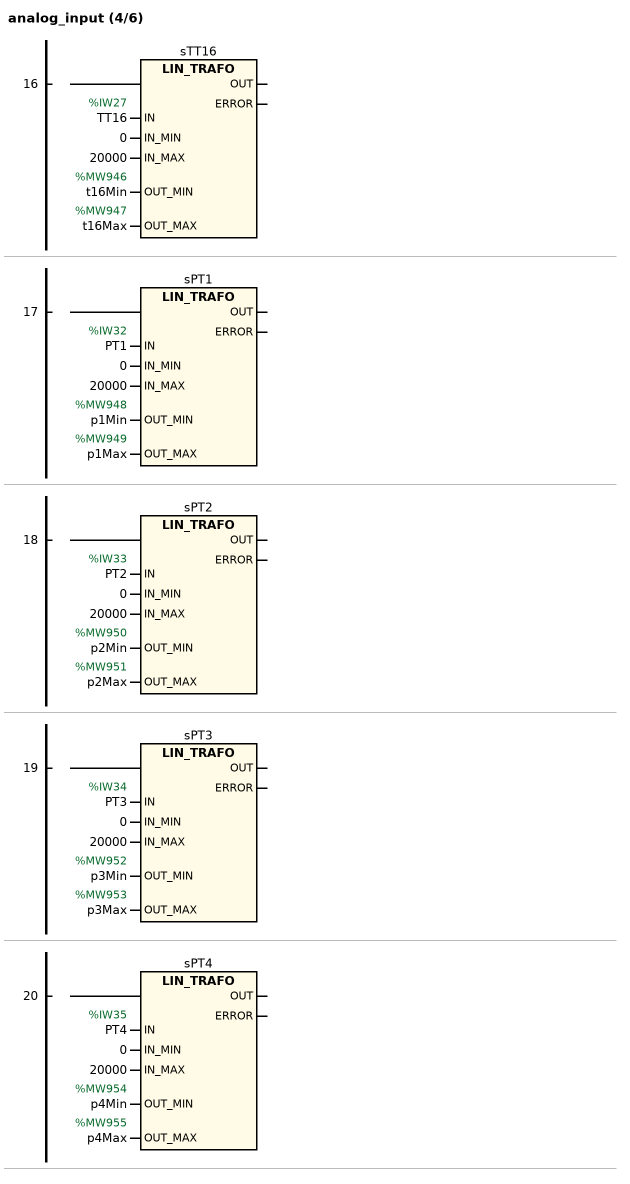
// NETWORK 16
//   TT16: A1_5 : | AT %IW27
//   t16Min: AT %MW946
//   t16Max: AT %MW947
sTT16(IN := TT16, IN_MIN := 0, IN_MAX := 20000, OUT_MIN := t16Min, OUT_MAX := t16Max); // LIN_TRAFO

// NETWORK 17
//   PT1: A1_6 : | AT %IW32
//   p1Min: AT %MW948
//   p1Max: AT %MW949
sPT1(IN := PT1, IN_MIN := 0, IN_MAX := 20000, OUT_MIN := p1Min, OUT_MAX := p1Max); // LIN_TRAFO

// NETWORK 18
//   PT2: A1_6 : | AT %IW33
//   p2Min: AT %MW950
//   p2Max: AT %MW951
sPT2(IN := PT2, IN_MIN := 0, IN_MAX := 20000, OUT_MIN := p2Min, OUT_MAX := p2Max); // LIN_TRAFO

// NETWORK 19
//   PT3: A1_6 : | AT %IW34
//   p3Min: AT %MW952
//   p3Max: AT %MW953
sPT3(IN := PT3, IN_MIN := 0, IN_MAX := 20000, OUT_MIN := p3Min, OUT_MAX := p3Max); // LIN_TRAFO

// NETWORK 20
//   PT4: A1_6 : | AT %IW35
//   p4Min: AT %MW954
//   p4Max: AT %MW955
sPT4(IN := PT4, IN_MIN := 0, IN_MAX := 20000, OUT_MIN := p4Min, OUT_MAX := p4Max); // LIN_TRAFO

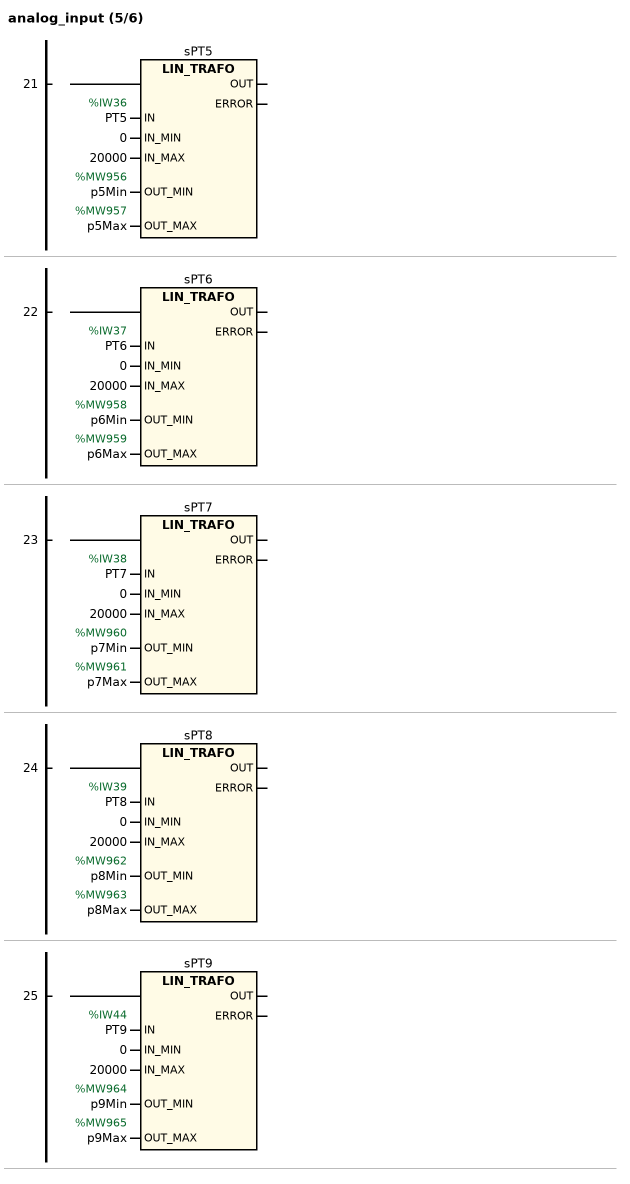
// NETWORK 21
//   PT5: A1_6 : | AT %IW36
//   p5Min: AT %MW956
//   p5Max: AT %MW957
sPT5(IN := PT5, IN_MIN := 0, IN_MAX := 20000, OUT_MIN := p5Min, OUT_MAX := p5Max); // LIN_TRAFO

// NETWORK 22
//   PT6: A1_6 : | AT %IW37
//   p6Min: AT %MW958
//   p6Max: AT %MW959
sPT6(IN := PT6, IN_MIN := 0, IN_MAX := 20000, OUT_MIN := p6Min, OUT_MAX := p6Max); // LIN_TRAFO

// NETWORK 23
//   PT7: A1_6 : | AT %IW38
//   p7Min: AT %MW960
//   p7Max: AT %MW961
sPT7(IN := PT7, IN_MIN := 0, IN_MAX := 20000, OUT_MIN := p7Min, OUT_MAX := p7Max); // LIN_TRAFO

// NETWORK 24
//   PT8: A1_6 : | AT %IW39
//   p8Min: AT %MW962
//   p8Max: AT %MW963
sPT8(IN := PT8, IN_MIN := 0, IN_MAX := 20000, OUT_MIN := p8Min, OUT_MAX := p8Max); // LIN_TRAFO

// NETWORK 25
//   PT9: A1_7 : | AT %IW44
//   p9Min: AT %MW964
//   p9Max: AT %MW965
sPT9(IN := PT9, IN_MIN := 0, IN_MAX := 20000, OUT_MIN := p9Min, OUT_MAX := p9Max); // LIN_TRAFO

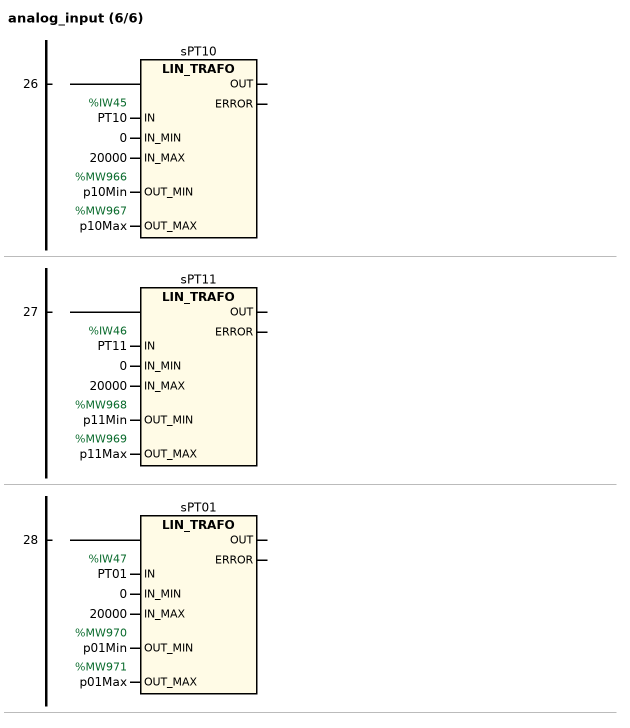
// NETWORK 26
//   PT10: A1_7 : | AT %IW45
//   p10Min: AT %MW966
//   p10Max: AT %MW967
sPT10(IN := PT10, IN_MIN := 0, IN_MAX := 20000, OUT_MIN := p10Min, OUT_MAX := p10Max); // LIN_TRAFO

// NETWORK 27
//   PT11: A1_7 : | AT %IW46
//   p11Min: AT %MW968
//   p11Max: AT %MW969
sPT11(IN := PT11, IN_MIN := 0, IN_MAX := 20000, OUT_MIN := p11Min, OUT_MAX := p11Max); // LIN_TRAFO

// NETWORK 28
//   PT01: A1_7 : | AT %IW47
//   p01Min: AT %MW970
//   p01Max: AT %MW971
sPT01(IN := PT01, IN_MIN := 0, IN_MAX := 20000, OUT_MIN := p01Min, OUT_MAX := p01Max); // LIN_TRAFO

END_PROGRAM

// MyController/Application/IN_A1_A12_A14_A17
PROGRAM IN_A1_A12_A14_A17
VAR


END_VAR

//ВХОДЫ А1========================================
DYMOHOD1_OPENED:=X1;
DYMOHOD1_CLOSED:= X2;
ZATVOR1_OPENED:= NOT X4;
ZATVOR1_CLOSED:= NOT X5;
DYMOHOD2_OPENED:= NOT X7;
DYMOHOD2_CLOSED:= NOT X8;
ZATVOR2_OPENED:=NOT X10;
ZATVOR2_CLOSED:=NOT X11;
FEEDER_OPENED:=NOT X13;
FEEDER_CLOSED:=NOT X14;
HVO_OPENED:= X16;
HVO_CLOSED:= X17;
PEREPUSK_OPENED:=X19;
PEREPUSK_CLOSED:=X20;
HEATER_OPENED:=X22;
HEATER_CLOSED:=X23;
//ВХОДЫ А1.1=====================================
ERR_PCH_PUMP_CYRCULATION:=not IX0;
ERR_PUMP1_CYRCULATION:=IX2;
ERR_PUMP2_CYRCULATION:=IX4;
ERR_PCH_PUMP1_NET:= NOT IX6;
ERR_PCH_PUMP2_NET:= NOT IX8;
ERR_M3_FEEDER:=IX10;
ERR_M4_FEEDER:=IX12;
VALVE_GAZ_OPENED:=IX15;
VALVE_GAZ_CLOSED:=IX16;
ERR_DEGAZATOR:=IX17;
FIRE:=IX18;
BREAKE:=IX19;
N0_SECURITY:=IX20;
SECURITY:=IX21;
BURNER1_WORKS:=IX22;
ERR_BURNER1:=IX23;
BURNER2_WORKS:=IX24;
ERR_BURNER2:=IX25;
ERR_GERM_BUR1:=IX26;//ГЕРМЕТИЧНОСТЬ ГОРЕЛКИ 1 НАРУШЕНА
BTN_HAND_MODE_PUMPS:=IX27;
BTN_AUTO_MODE_PUMPS:=IX28;
BTN_HAND_MODE_BOILERS:=IX29;
BTN_AUTO_MODE_BOILERS:=IX30;
BTN_HAND_MODE_VALVES:=IX31;
//ВХОДЫ А1.2=====================================
BTN_AUTO_MODE_VALVES:=IIX0;
ERR_GAZ:=NOT IIX1;

BURNER2_IN_AUTO_MODE:=IIX6;
ERR_GERM_BURNER2:=IIX7;
RKF:=NOT IIX12;
BURNER1_IN_AUTO_MODE:=IIX15;

//АНАЛОГОВЫЕ ВХОДЫ А1.4-A1.7==========================
TT1_DYMA_1:=REAL_TO_INT(analog_input.sTT1.OUT);     //ТЕЬПЕРАТУРА ДЫМА ЗА КОТЛОМ 1
TT2_WTR_IN_1:=REAL_TO_INT(analog_input.sTT2.OUT);    //ТЕМПЕРАТУРА СЕТЕВОЙ ВОДЫ ПРЕД КОТЛОМ 1
TT3_WTR_OUT_1:=REAL_TO_INT(analog_input.sTT3.OUT);    //ТЕМПЕРАТУРА ОБРАТНОЙ СЕТЕВОЙ ВОДЫ НА ВЫХОДЕ ИЗ КОТЛА 1
TT4_DYMA_UTIL_OUT:=REAL_TO_INT(analog_input.sTT4.OUT);//ТЕМПЕРАТУРА ДЫМА ЗА УТИЛИЗАТОРОМ
TT5_DYMA_2:=REAL_TO_INT(analog_input.sTT5.OUT);      //ТЕМПЕРАТУРА ДЫМА ЗА КОТЛОМ 2
TT6_WTR_UTIL_IN:=REAL_TO_INT(analog_input.sTT6.OUT);//ТЕМПЕРАТУРА СЕТЕВОЙ ВОДЫ ПЕРЕД УТИЛИЗАТОРОМ
TT7_WTR_IN_2:=REAL_TO_INT(analog_input.sTT7.OUT);    //ТЕМПЕРАТУРА ОБРАТНОЙ ВОДЫ ПЕРЕД КОТЛОМ 2
TT8_WTR_OUT_2:=REAL_TO_INT(analog_input.sTT8.OUT);   //ТЕМПЕРАТУРА ОБРАТНОЙ ВОДЫ ПОСЛЕ КОТЛА 2
TT9_WTR_IN_3H:=REAL_TO_INT(analog_input.sTT9.OUT)    ;//ТЕМПЕРАТУРА СЕТЕВОЙ ВОДЫ ПЕРЕД ТРЕХХОДОВЫМ ПОДМЕСА
TT10_WTR_OUT_3H:=REAL_TO_INT(analog_input.sTT10.OUT);//ТЕМПЕРАТУРА СЕТЕВОЙ ВОДЫ ПОСЛЕ ТРЕХХОДОВОГО ПОДМЕСА
TT11_NET_WTR_IN1:=REAL_TO_INT(analog_input.sTT11.OUT);//ТЕМПЕРАТУРА СЕТЕВОЙ ВОДЫ ПЕРЕД КОТЛАМИ
TT12_NET_WTR_OUT:=REAL_TO_INT(analog_input.sTT12.OUT);//ТЕМПЕРАТУРА ПРЯМОЙ СЕТЕВОЙ ВОДЫ НА ВЫХОДЕ ИЗ КОТЕЛЬНОЙ
TT13_NET_WTR_IN2:=REAL_TO_INT(analog_input.sTT13.OUT);//ТЕМПЕРАТУРА ОБРАТНОЙ СЕТЕВОЙ ВОДЫ НА ВХОДЕ В КОТЕЛЬНУЮ
TT14_WTR_FEDER:=REAL_TO_INT(analog_input.sTT14.OUT);  //ТЕМПЕРАТУРА ПРЯМОЙ СЕТЕВОЙ ВОДЫ НА ВВОДЕ В КОТЕЛЬНУЮ
TT15_IN_ROOM:=REAL_TO_INT(analog_input.sTT15.OUT);   //ТЕМПЕРАТУРА В КОТЕЛЬНОЙ
TT16_ON_AIR:=REAL_TO_INT(analog_input.sTT16.OUT);    //ТЕМПЕРАТУРА НА УЛИЦЕ
PT1_WTR_IN_1:=REAL_TO_INT(analog_input.sPT1.OUT);    //ДАВЛЕНИЕ ОБРАТНОЙ СЕТЕВОЙ ВОДЫ ПЕРЕД КОТЛОМ 1
PT2_WTR_OUT_1:=REAL_TO_INT(analog_input.sPT2.OUT);    //ДАВЛЕНИЕ ОБРАТНОЙ СЕТЕВОЙ ВОДЫ ПОСЛЕ КОТЛА 1
PT3_WTR_UTIL_IN:=REAL_TO_INT(analog_input.sPT3.OUT); //ДАВЛЕНИЕ ОБРАТНОЙ СЕТЕВОЙ ВОДЫ ПЕРЕД УТИЛИЗАТОРОМ 
PT4_WTR_IN_2:=REAL_TO_INT(analog_input.sPT4.OUT);    //ДАВЛЕНИЕ ОБРАТНОЙ СЕТЕВОЙ ВОДЫ ПЕРЕД КОТЛОМ 2
PT5_WTR_OUT_2:=REAL_TO_INT(analog_input.sPT5.OUT);   //ДАВЛЕНИЕ ОБРАТНОЙ СЕТЕВОЙ ВОДЫ ПОСЛЕ КОТЛА 2
PT6_WTR_IN_3H:=REAL_TO_INT(analog_input.sPT6.OUT);   //ДАВЛЕНИЕ СЕТЕВОЙ ВОДЫ ПЕРЕД ТРЕХХОДОВЫМ ПОДМЕСА
PT7_WTR_OUT_3H:=REAL_TO_INT(analog_input.sPT7.OUT);  //ДАВЛЕНИЕ СЕТЕВОЙ ВОДЫ ПОСЛЕ ТРЕХХОДОВОГО ПОДМЕСА
PT8_WTR_OUT_BOILER:=REAL_TO_INT(analog_input.sPT8.OUT);//ДАВЛЕНИЕ СЕТЕВОЙ ВОДЫ НА ВЫХОДЕ ИЗ КОТЕЛЬНОЙ
PT9_WTR_IN_BOILER:=REAL_TO_INT(analog_input.sPT9.OUT);//ДАВЛЕНИЕ СЕТЕВОЙ ВОДЫ НА ВХОДЕ В КОТЕЛЬНУЮ
PT10_LEVEL_HVO:=REAL_TO_INT(analog_input.sPT10.OUT);  //УРОВЕНЬ В БАКЕ ХВО
PT11_WTR_IN_BOILER:=REAL_TO_INT(analog_input.sPT11.OUT);//ДАВЛЕНИЕ ИСХОДНОЙ ВОДЫ НА ВВОДЕ В КОТЕЛЬНУЮ
PT01_GAZ:=REAL_TO_INT(analog_input.sPT01.OUT);        //ДАВЛЕНИЕ ГАЗА

END_PROGRAM

// MyController/Application/MB_IN
PROGRAM MB_IN
VAR
END_VAR

(*
TBTN_ON_SMALL_FLAME_BURNER_1:=MW204.2;
TBTN_ON_LAGE_FLAME_BURNER_1:=MW204.3;
TBTN_ON_SMALL_FLAME_BURNER_2:=MW204.4;
TBTN_ON_LAGE_FLAME_BURNER_2:=MW204.5;

BTN_OPEN_DYMOHOD1:=MW205.0;
BTN_CLOSE_DYMOHOD1:=MW205.1;
BTN_OPEN_ZATVOR1:=MW205.2;
BTN_CLOSE_ZATVOR1:=MW205.3;
BTN_OPEN_DYMOHOD2:=MW205.4;
BTN_CLOSE_DYMOHOD2:=MW205.5;
BTN_OPEN_ZATVOR2:=MW205.6;
BTN_CLOSE_ZATVOR2:=MW205.7;
BTN_OPEN_FEEDER:=MW205.8;
BTN_CLOSE_FEEDER:=MW205.9;
BTN_OPEN_HVO:=MW205.10;
BTN_CLOSE_HVO:=MW205.11;
BTN_OPEN_PEREPUSK:=MW205.12;
BTN_CLOSE_PEREPUSK:=MW205.13;
BTN_OPEN_HEATER:=MW205.14;
BTN_CLOSE_HEATER:=MW205.15;

BTN_RUN_PUMP_CYRCULATION:=MW206.0;
BTN_RUN_PUMP_CYRCULATION1:=MW206.1;
BTN_RUN_PUMP_CYRCULATION2:=MW206.2;
BTN_RUN_PUMP1_NET:=MW206.3;
BTN_RUN_PUMP2_NET:=MW206.4;
BTN_RUN_M3_FEEDER:=MW206.5;
BTN_RUN_M4_FEEDER:=MW206.6;
BTN_OPEN_GAZ:=MW206.7;
BTN_CLOSE_GAZ:=MW206.8;
BTN_RUN_SIGNAL_FIRE:=MW206.9;
//BTN_RUN_SIGNAL_BREAKE:=MW206.10;
//RESET_ERR:=MW206.11;
//PRIOR_BOILER_1:=MW206.12;
//PRIOR_BOILER_2:=MW206.13;
//PRIOR_PUMP_M5:=MW206.14;
//AUTO_MODE:=MW206.15;

//PRIOR_PUMP_M6:=MW211.0;
//PRIOR_PUMP_M1:=MW211.1;
//PRIOR_PUMP_M2:=MW211.2;
//BTN_PUSK_STOP_BOILER:=MW211.3;

resv_data_from_flowmtr_ADR6[6]:=0;
resv_data_from_flowmtr_ADR6[7]:=0;
resv_data_from_flowmtr_ADR6[8]:=0;
resv_data_from_flowmtr_ADR6[9]:=0;

resv_data_from_flowmtr_ADR7[6]:=0;
resv_data_from_flowmtr_ADR7[7]:=0;
resv_data_from_flowmtr_ADR7[8]:=0;
resv_data_from_flowmtr_ADR7[9]:=0;

resv_data_from_flowmtr_ADR8[6]:=0;
resv_data_from_flowmtr_ADR8[7]:=0;
resv_data_from_flowmtr_ADR8[8]:=0;
resv_data_from_flowmtr_ADR8[9]:=0;*)

END_PROGRAM

// MyController/Application/get_data_from_CKM
PROGRAM get_data_from_CKM
VAR
	good: BOOL;
	t: INT;
END_VAR

skm_number := skm_number_arr[0]*65536+skm_number_arr[1];
FOR t:=0 TO 37 DO
	skm_all_mw[2*t] := skm_all[2*t+1];
	skm_all_mw[2*t+1] := skm_all[2*t];
END_FOR

(*IF step=3 THEN
	resv_data_from_ckm[0]:=0;
	
	data_to_send[0]:=16#10;
	data_to_send[1]:=16#40;
	data_to_send[2]:=16#00;
	data_to_send[3]:=data_to_send[1]+data_to_send[2];
	data_to_send[4]:=16#16;
	
	IF resv_data_from_ckm[0]=16#E5
	THEN	step:=step+1;
	ELSE	step:=3;
	END_IF 		
END_IF

IF (step=4) THEN
	resv_data_from_ckm[0]:=0;
	
	data_to_send[0]:=16#68;
	data_to_send[1]:=16#04;
	data_to_send[2]:=16#04;
	data_to_send[3]:=16#68;
	data_to_send[4]:=16#53;
	data_to_send[5]:=16#00;
	data_to_send[6]:=16#50;
	data_to_send[7]:=16#10;
	data_to_send[8]:=data_to_send[4]+data_to_send[5]+data_to_send[6]+data_to_send[7];
	data_to_send[9]:=16#16;

	//good:= send_to_ckm(10,1);
	
	IF resv_data_from_ckm[0]=16#E5
	THEN	step:=step+1;
	ELSE	step:=3;
	END_IF 		
END_IF

IF (step=5) THEN
	
	data_to_send[0]:=16#10;
	data_to_send[1]:=16#5B;
	data_to_send[2]:=16#00;
	data_to_send[3]:=data_to_send[1]+data_to_send[2];
	data_to_send[4]:=16#16;

	//good:= send_to_ckm(4,118);
	
	
	RASHOD_WATER:=resv_data_from_ckm[50];
	RASHOD_WATER:=SHL(RASHOD_WATER,8)+resv_data_from_ckm[51];
	step:=0;		
		
END_IF
*)

END_PROGRAM

// MyController/Application/FB/send_to_ckm
FUNCTION send_to_ckm : BOOL;
VAR_INPUT
	QuantityToSend: UINT;
	SizeRecv: UINT;
	M1: BOOL;
END_VAR
VAR
	send_data_to_oven: SEND_RECV_MSG;
	send_data_to_skm: SEND_RECV_MSG;
	SL_1: ADDRESS;
	ADDRES_COM: ADDM;
END_VAR

VAR_OUTPUT
	good: BOOL;
END_VAR

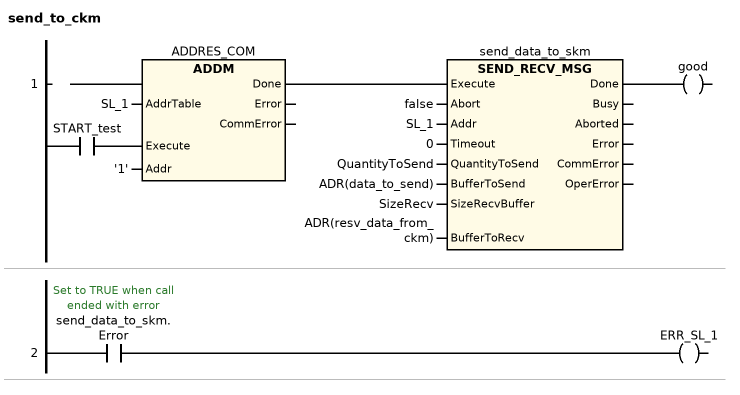
// NETWORK 1
ADDRES_COM(AddrTable := SL_1, Execute := START_test, Addr := '1'); // ADDM
send_data_to_skm(
    Execute := ADDRES_COM.Done,
    Abort := false,
    Addr := SL_1,
    Timeout := 0,
    QuantityToSend := QuantityToSend,
    BufferToSend := ADR(data_to_send),
    SizeRecvBuffer := SizeRecv,
    BufferToRecv := ADR(resv_data_from_ckm)); // SEND_RECV_MSG
good := send_data_to_skm.Done;

// NETWORK 2
//   send_data_to_skm.Error: Set to TRUE when call ended with error
ERR_SL_1 := send_data_to_skm.Error;

END_FUNCTION

// MyController/Application/reset_flowmetr
PROGRAM reset_flowmetr
VAR
	BLINK_RESET_FLOW : BLINK;
	RISE_IMPUT_FLOW : R_TRIG;
	good: BOOL;
END_VAR

VAR_OUTPUT
	zero_flow: BOOL;
END_VAR

//Каждые TIMELOW секунд сбрасываем массив приема данных из счетчиков на тот случай если связь пропадет
BLINK_RESET_FLOW(ENABLE:=1,TIMELOW:=T#30S,TIMEHIGH:=T#2S);
RISE_IMPUT_FLOW(CLK:=BLINK_RESET_FLOW.OUT); 
zero_flow:=BLINK_RESET_FLOW.OUT;
IF RISE_IMPUT_FLOW.Q=1 THEN
	resv_data_from_flowmtr_ADR6[6]:=0;
	resv_data_from_flowmtr_ADR6[7]:=0;
	resv_data_from_flowmtr_ADR6[8]:=0;
	resv_data_from_flowmtr_ADR6[9]:=0;

	resv_data_from_flowmtr_ADR7[6]:=0;
	resv_data_from_flowmtr_ADR7[7]:=0;
	resv_data_from_flowmtr_ADR7[8]:=0;
	resv_data_from_flowmtr_ADR7[9]:=0;

	resv_data_from_flowmtr_ADR8[6]:=0;
	resv_data_from_flowmtr_ADR8[7]:=0;
	resv_data_from_flowmtr_ADR8[8]:=0;
	resv_data_from_flowmtr_ADR8[9]:=0;
END_IF

END_PROGRAM

// MyController/Application/send_data_to_flowmeter
PROGRAM send_data_to_flowmeter
VAR
	SL_1: ADDRESS;
	ADDRES_COM: ADDM;
	add_step: BLINK;
	M1: BOOL;
END_VAR
VAR // added by the converter: edge detectors and wires of the graphical bodies
    _rt1 : R_TRIG;
    _ft1, _ft2 : F_TRIG;
END_VAR

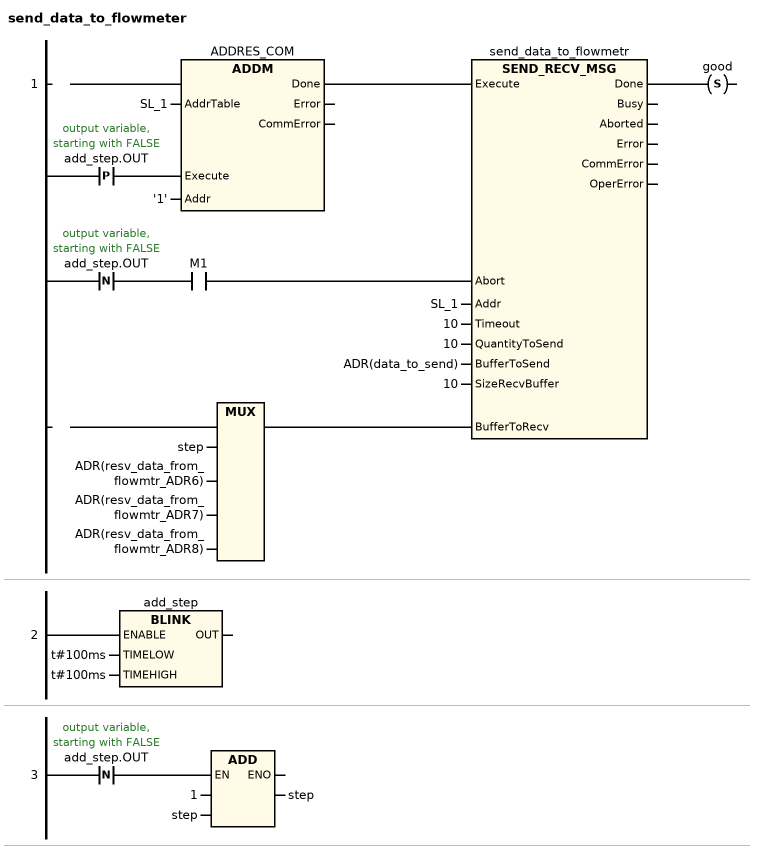
// NETWORK 1
//   add_step.OUT: output variable, starting with FALSE
//   step: БЛОК ДЛЯ ОБМЕНА С РАСХОДОМЕРОМ ======КОЕЦ====== БЛОК ДЛЯ ОБМЕНА С ОВЕНОМ ======НАЧАЛО======
_rt1(CLK := add_step.OUT);
ADDRES_COM(AddrTable := SL_1, Execute := _rt1.Q, Addr := '1'); // ADDM
_ft1(CLK := add_step.OUT);
send_data_to_flowmetr(
    Execute := ADDRES_COM.Done,
    Abort := _ft1.Q AND M1,
    Addr := SL_1,
    Timeout := 10,
    QuantityToSend := 10,
    BufferToSend := ADR(data_to_send),
    SizeRecvBuffer := 10,
    BufferToRecv := MUX(step, ADR(resv_data_from_flowmtr_ADR6), ADR(resv_data_from_flowmtr_ADR7), ADR(resv_data_from_flowmtr_ADR8))); // SEND_RECV_MSG
good S= send_data_to_flowmetr.Done;

// NETWORK 2
add_step(ENABLE := TRUE, TIMELOW := t#100ms, TIMEHIGH := t#100ms); // BLINK

// NETWORK 3
//   add_step.OUT: output variable, starting with FALSE
//   step: БЛОК ДЛЯ ОБМЕНА С РАСХОДОМЕРОМ ======КОЕЦ====== БЛОК ДЛЯ ОБМЕНА С ОВЕНОМ ======НАЧАЛО======
_ft2(CLK := add_step.OUT);
IF _ft2.Q THEN step := 1 + step; END_IF

END_PROGRAM

// MyController/Application/A_TESTS/zadanie_for_m1_m2
PROGRAM zadanie_for_m1_m2
VAR
	ZADANIE_FOR_PCH_M1_M2: INT;
	e: INT;
END_VAR

(*IF PT8_WTR_OUT_BOILER<PT8_WTR_OUT_BOILER_ZADANIE
	THEN IF ZADANIE_FOR_PCH_M1_M2<500
			THEN ZADANIE_FOR_PCH_M1_M2:=ZADANIE_FOR_PCH_M1_M2+1;
		END_IF
	
	ELSE IF ZADANIE_FOR_PCH_M1_M2>0
			THEN ZADANIE_FOR_PCH_M1_M2:=ZADANIE_FOR_PCH_M1_M2-1;
		END_IF
END_IF



IF AUTO_MODE=1
	THEN PCH_PUMP_M1_ZADANIE:=ZADANIE_FOR_PCH_M1_M2;
		PCH_PUMP_M2_ZADANIE:=ZADANIE_FOR_PCH_M1_M2;
	ELSE PCH_PUMP_M1_ZADANIE:=MANUAL_ZADANIE_FOR_PCH;
		PCH_PUMP_M2_ZADANIE:=MANUAL_ZADANIE_FOR_PCH;
END_IF
*)

END_PROGRAM

// A_TESTS/zadanie_for_m1_m2
PROGRAM zadanie_for_m1_m2
VAR
	ZADANIE_FOR_PCH_M1_M2: INT;
	e: INT;
END_VAR

(*IF PT8_WTR_OUT_BOILER<PT8_WTR_OUT_BOILER_ZADANIE
	THEN IF ZADANIE_FOR_PCH_M1_M2<500
			THEN ZADANIE_FOR_PCH_M1_M2:=ZADANIE_FOR_PCH_M1_M2+1;
		END_IF
	
	ELSE IF ZADANIE_FOR_PCH_M1_M2>0
			THEN ZADANIE_FOR_PCH_M1_M2:=ZADANIE_FOR_PCH_M1_M2-1;
		END_IF
END_IF



IF AUTO_MODE=1
	THEN PCH_PUMP_M1_ZADANIE:=ZADANIE_FOR_PCH_M1_M2;
		PCH_PUMP_M2_ZADANIE:=ZADANIE_FOR_PCH_M1_M2;
	ELSE PCH_PUMP_M1_ZADANIE:=MANUAL_ZADANIE_FOR_PCH;
		PCH_PUMP_M2_ZADANIE:=MANUAL_ZADANIE_FOR_PCH;
END_IF
*)

END_PROGRAM

// MyController/Application/get_data_from_flowmetr
PROGRAM get_data_from_flowmetr
VAR
	good: BOOL;
	man: INT;
END_VAR

IF step<=0 OR step>=3 THEN
	step:= 0;	
END_IF

IF step=0 THEN
//ПОЛУЧЕНИЕ ТЕКУЩЕГО РАСХОДА, СЧЕТЧИК С АДРЕСОМ 6 BOILER 1
	data_to_send[0]:=16#55;//признак начала пакета
	data_to_send[1]:=16#06;//адрес 
	data_to_send[2]:=16#F9;//инверсия адреса
	data_to_send[3]:=16#0C;//группа команд
	data_to_send[4]:=16#01;//чтение из памяти 2 К таймера
	data_to_send[5]:=16#03;//число байт посылаемых данных
	data_to_send[6]:=16#00;//старший байт начального адреса
	data_to_send[7]:=16#B4;//младший байт начального адреса
	data_to_send[8]:=16#04;//количество читаемых байт
	data_to_send[9]:=16#E3;//контрольная сумма not(b1+....+bn)
	IF reset_flowmetr.zero_flow=0 THEN
		FL_BOILER_1:=resv_data_from_flowmtr_ADR6[6];
		FL_BOILER_1:=SHL (FL_BOILER_1, 8);
		FL_BOILER_1:=FL_BOILER_1+resv_data_from_flowmtr_ADR6[7];
		FL_BOILER_1:=SHL (FL_BOILER_1, 8);
		FL_BOILER_1:=FL_BOILER_1+resv_data_from_flowmtr_ADR6[8];
  		FL_BOILER_1:=SHL (FL_BOILER_1, 8);
		FL_BOILER_1:=FL_BOILER_1+resv_data_from_flowmtr_ADR6[9];
	END_IF
	//step:=step+1;
END_IF

IF step=1 THEN
//ПОЛУЧЕНИЕ ТЕКУЩЕГО РАСХОДА, СЧЕТЧИК С АДРЕСОМ 7 BOILER 2
	data_to_send[0]:=16#55;//признак начала пакета
	data_to_send[1]:=16#07;//адрес 
	data_to_send[2]:=16#F8;//инверсия адреса
	data_to_send[3]:=16#0C;//группа команд
	data_to_send[4]:=16#01;//чтение из памяти 2 К таймера
	data_to_send[5]:=16#03;//число байт посылаемых данных
	data_to_send[6]:=16#00;//старший байт начального адреса
	data_to_send[7]:=16#B4;//младший байт начального адреса
	data_to_send[8]:=16#04;//количество читаемых байт
	data_to_send[9]:=16#E3;//контрольная сумма not(b1+....+bn)
	IF reset_flowmetr.zero_flow=0 THEN
		FL_BOILER_2:=resv_data_from_flowmtr_ADR7[6];
		FL_BOILER_2:=SHL (FL_BOILER_2, 8);
		FL_BOILER_2:=FL_BOILER_2+resv_data_from_flowmtr_ADR7[7];
		FL_BOILER_2:=SHL (FL_BOILER_2, 8);
		FL_BOILER_2:=FL_BOILER_2+resv_data_from_flowmtr_ADR7[8];
  		FL_BOILER_2:=SHL (FL_BOILER_2, 8);
		FL_BOILER_2:=FL_BOILER_2+resv_data_from_flowmtr_ADR7[9];
		//FL_BOILER_2:=0;
	END_IF
	//step:=step+1;
END_IF


IF step=2 THEN
//ПОЛУЧЕНИЕ ТЕКУЩЕГО РАСХОДА СЧЕТЧИК С АДРЕСОМ 8 GAZ
	data_to_send[0]:=16#55;//признак начала пакета
	data_to_send[1]:=16#08;//адрес 
	data_to_send[2]:=16#F7;//инверсия адреса
	data_to_send[3]:=16#0C;//группа команд
	data_to_send[4]:=16#01;//чтение из памяти 2 К таймера
	data_to_send[5]:=16#03;//число байт посылаемых данных
	data_to_send[6]:=16#00;//старший байт начального адреса
	data_to_send[7]:=16#B4;//младший байт начального адреса
	data_to_send[8]:=16#04;//количество читаемых байт
	data_to_send[9]:=16#E3;//контрольная сумма not(b1+....+bn)
	IF reset_flowmetr.zero_flow=0 THEN
		FL_HVO:=resv_data_from_flowmtr_ADR8[6];
		FL_HVO:=SHL (FL_HVO, 8);
		FL_HVO:=FL_HVO + resv_data_from_flowmtr_ADR8[7];
		FL_HVO:=SHL (FL_HVO, 8);
		FL_HVO:=FL_HVO + resv_data_from_flowmtr_ADR8[8];
  		FL_HVO:=SHL (FL_HVO, 8);
		FL_HVO:=FL_HVO + resv_data_from_flowmtr_ADR8[9];
	END_IF
	//step:=step+1;
END_IF

END_PROGRAM

// MyController/Application/BURNERS_GAZ_GRU
PROGRAM BURNERS_GAZ_GRU
VAR
	TM_CLOSE_ZATVOR_1: TOF;
	GAZ_GRU_CYCLE_OPEN: BOOL;
	GAZ_GRU_CYCLE_CLOSE: BOOL;
	TM_CLOSE_GAZ_GRU: TOF;	

	tm_eer_prod1: TON;
	tm_err_wiring1: TON;
	tm_err_cold1: TON;
	
	tm_eer_prod2: TON;
	tm_err_wiring2: TON;
	tm_err_cold2: TON;
	
	
	tm_pt01_gaz: TON;
	//ERR_BURNER_1: BOOL;
	tm_pt1: TON;
	tm_pt2: TON;
	tm_pt4: TON;
END_VAR

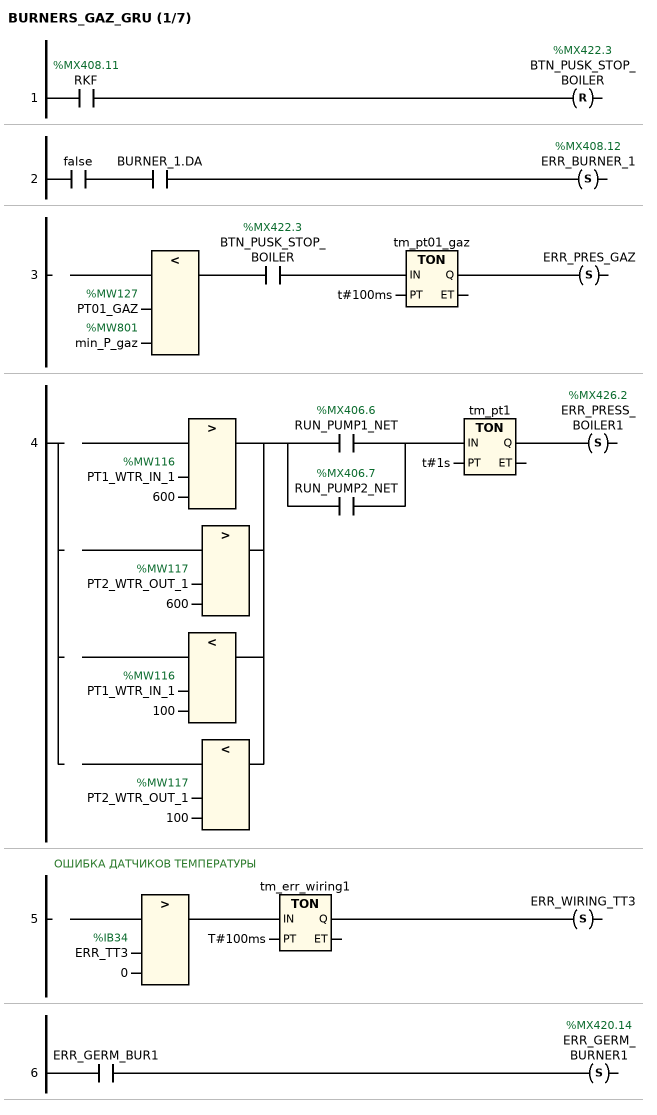
// NETWORK 1
//   RKF: AT %MX408.11
//   BTN_PUSK_STOP_BOILER: AT %MX422.3
BTN_PUSK_STOP_BOILER R= RKF;

// NETWORK 2
//   ERR_BURNER_1: AT %MX408.12
ERR_BURNER_1 S= false AND BURNER_1.DA;

// NETWORK 3
//   PT01_GAZ: AT %MW127
//   min_P_gaz: AT %MW801
//   BTN_PUSK_STOP_BOILER: AT %MX422.3
tm_pt01_gaz(IN := PT01_GAZ < min_P_gaz AND BTN_PUSK_STOP_BOILER, PT := t#100ms); // TON
ERR_PRES_GAZ S= tm_pt01_gaz.Q;

// NETWORK 4
//   tm_pt1: ERR_BURNER_1: BOOL;
//   PT1_WTR_IN_1: AT %MW116
//   PT2_WTR_OUT_1: AT %MW117
//   RUN_PUMP1_NET: AT %MX406.6
//   RUN_PUMP2_NET: AT %MX406.7
//   ERR_PRESS_BOILER1: AT %MX426.2
tm_pt1(IN := (PT1_WTR_IN_1 > 600 OR PT2_WTR_OUT_1 > 600 OR PT1_WTR_IN_1 < 100 OR PT2_WTR_OUT_1 < 100) AND (RUN_PUMP1_NET OR RUN_PUMP2_NET), PT := t#1s); // TON
ERR_PRESS_BOILER1 S= tm_pt1.Q;

// NETWORK 5
// ОШИБКА ДАТЧИКОВ ТЕМПЕРАТУРЫ
//   ERR_TT3: A1_4 : | AT %IB34
tm_err_wiring1(IN := ERR_TT3 > 0, PT := T#100ms); // TON
ERR_WIRING_TT3 S= tm_err_wiring1.Q;

// NETWORK 6
//   ERR_GERM_BURNER1: AT %MX420.14
ERR_GERM_BURNER1 S= ERR_GERM_BUR1;

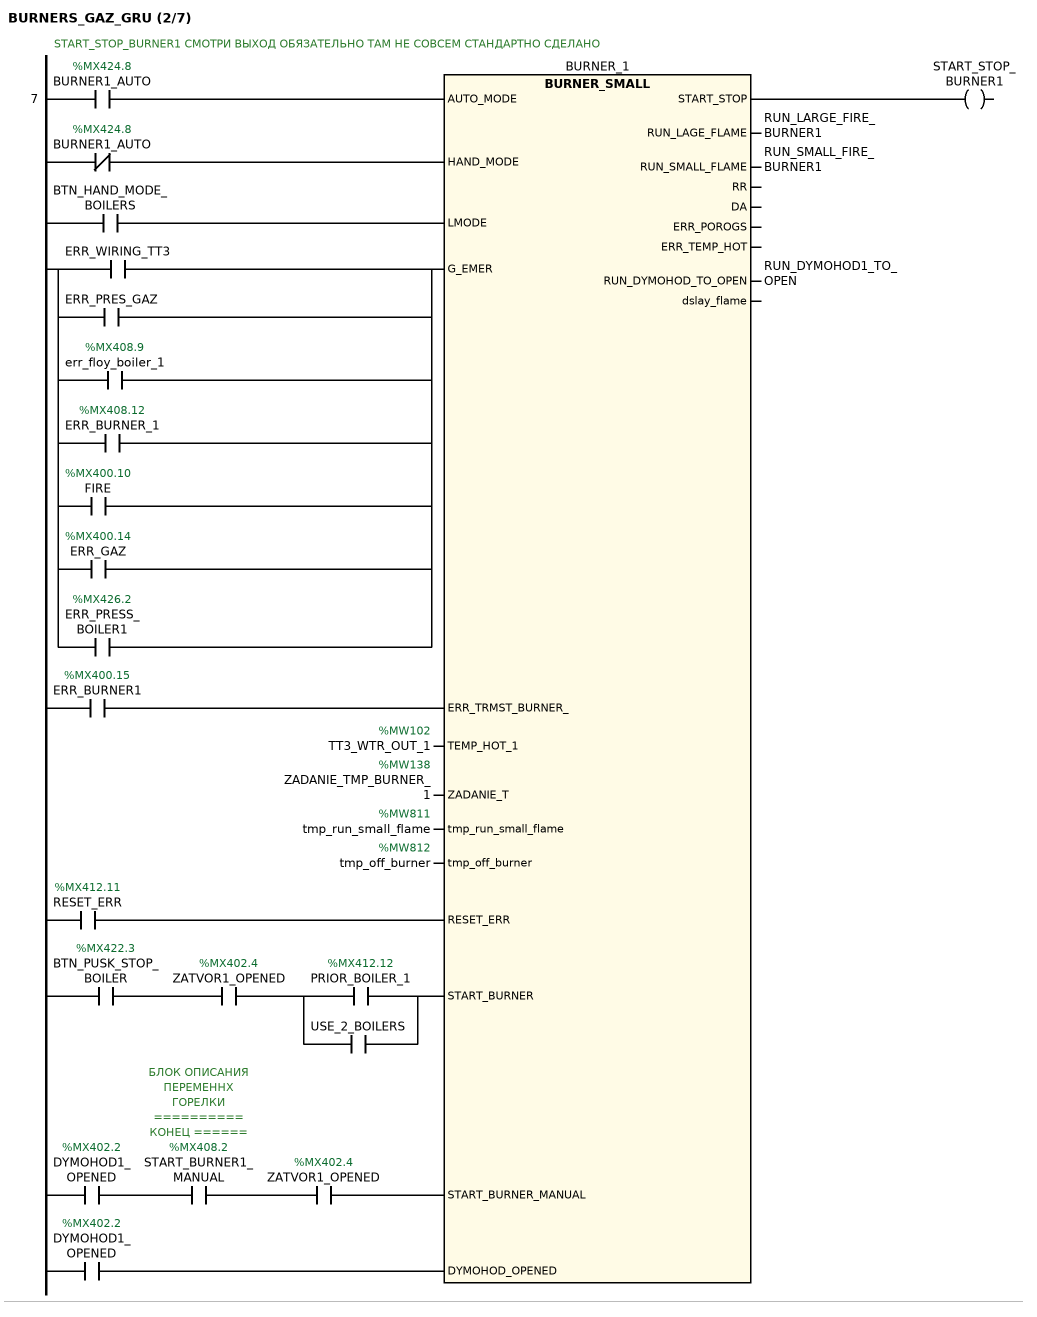
// NETWORK 7
// START_STOP_BURNER1 СМОТРИ ВЫХОД ОБЯЗАТЕЛЬНО ТАМ НЕ СОВСЕМ СТАНДАРТНО СДЕЛАНО
//   BURNER1_AUTO: AT %MX424.8
//   err_floy_boiler_1: AT %MX408.9
//   ERR_BURNER_1: AT %MX408.12
//   FIRE: AT %MX400.10
//   ERR_GAZ: AT %MX400.14
//   ERR_PRESS_BOILER1: AT %MX426.2
//   ERR_BURNER1: AT %MX400.15
//   TT3_WTR_OUT_1: AT %MW102
//   ZADANIE_TMP_BURNER_1: AT %MW138
//   tmp_run_small_flame: AT %MW811
//   tmp_off_burner: AT %MW812
//   RESET_ERR: AT %MX412.11
//   BTN_PUSK_STOP_BOILER: AT %MX422.3
//   ZATVOR1_OPENED: AT %MX402.4
//   PRIOR_BOILER_1: AT %MX412.12
//   DYMOHOD1_OPENED: AT %MX402.2
//   START_BURNER1_MANUAL: БЛОК ОПИСАНИЯ ПЕРЕМЕННХ ГОРЕЛКИ ========== КОНЕЦ ====== | AT %MX408.2
//   RUN_LARGE_FIRE_BURNER1: AT %MX406.15
//   RUN_SMALL_FIRE_BURNER1: AT %MX406.14
BURNER_1(
    AUTO_MODE := BURNER1_AUTO,
    HAND_MODE := NOT BURNER1_AUTO,
    LMODE := BTN_HAND_MODE_BOILERS,
    G_EMER := ERR_WIRING_TT3 OR ERR_PRES_GAZ OR err_floy_boiler_1 OR ERR_BURNER_1 OR FIRE OR ERR_GAZ OR ERR_PRESS_BOILER1,
    ERR_TRMST_BURNER_ := ERR_BURNER1,
    TEMP_HOT_1 := TT3_WTR_OUT_1,
    ZADANIE_T := ZADANIE_TMP_BURNER_1,
    tmp_run_small_flame := tmp_run_small_flame,
    tmp_off_burner := tmp_off_burner,
    RESET_ERR := RESET_ERR,
    START_BURNER := BTN_PUSK_STOP_BOILER AND ZATVOR1_OPENED AND (PRIOR_BOILER_1 OR USE_2_BOILERS),
    START_BURNER_MANUAL := DYMOHOD1_OPENED AND START_BURNER1_MANUAL AND ZATVOR1_OPENED,
    DYMOHOD_OPENED := DYMOHOD1_OPENED,
    RUN_LAGE_FLAME => RUN_LARGE_FIRE_BURNER1,
    RUN_SMALL_FLAME => RUN_SMALL_FIRE_BURNER1,
    RUN_DYMOHOD_TO_OPEN => RUN_DYMOHOD1_TO_OPEN); // BURNER_SMALL
START_STOP_BURNER1 := BURNER_1.START_STOP;

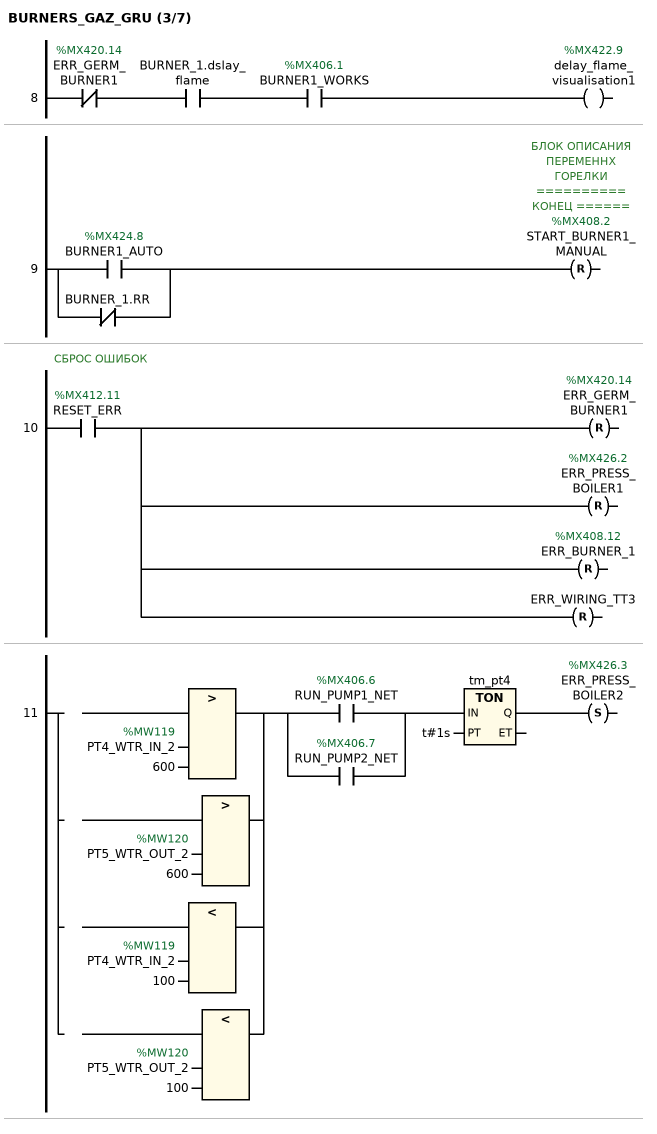
// NETWORK 8
//   ERR_GERM_BURNER1: AT %MX420.14
//   BURNER1_WORKS: AT %MX406.1
//   delay_flame_visualisation1: AT %MX422.9
delay_flame_visualisation1 := NOT ERR_GERM_BURNER1 AND BURNER_1.dslay_flame AND BURNER1_WORKS;

// NETWORK 9
//   BURNER1_AUTO: AT %MX424.8
//   START_BURNER1_MANUAL: БЛОК ОПИСАНИЯ ПЕРЕМЕННХ ГОРЕЛКИ ========== КОНЕЦ ====== | AT %MX408.2
START_BURNER1_MANUAL R= BURNER1_AUTO OR NOT BURNER_1.RR;

// NETWORK 10
// СБРОС ОШИБОК
//   RESET_ERR: AT %MX412.11
//   ERR_GERM_BURNER1: AT %MX420.14
//   ERR_PRESS_BOILER1: AT %MX426.2
//   ERR_BURNER_1: AT %MX408.12
ERR_GERM_BURNER1 R= RESET_ERR;
ERR_PRESS_BOILER1 R= RESET_ERR;
ERR_BURNER_1 R= RESET_ERR;
ERR_WIRING_TT3 R= RESET_ERR;

// NETWORK 11
//   PT4_WTR_IN_2: AT %MW119
//   PT5_WTR_OUT_2: AT %MW120
//   RUN_PUMP1_NET: AT %MX406.6
//   RUN_PUMP2_NET: AT %MX406.7
//   ERR_PRESS_BOILER2: AT %MX426.3
tm_pt4(IN := (PT4_WTR_IN_2 > 600 OR PT5_WTR_OUT_2 > 600 OR PT4_WTR_IN_2 < 100 OR PT5_WTR_OUT_2 < 100) AND (RUN_PUMP1_NET OR RUN_PUMP2_NET), PT := t#1s); // TON
ERR_PRESS_BOILER2 S= tm_pt4.Q;

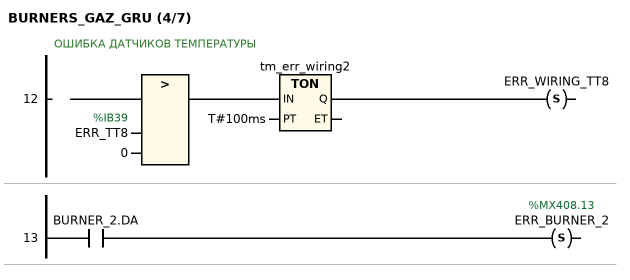
// NETWORK 12
// ОШИБКА ДАТЧИКОВ ТЕМПЕРАТУРЫ
//   ERR_TT8: A1_4 : | AT %IB39
tm_err_wiring2(IN := ERR_TT8 > 0, PT := T#100ms); // TON
ERR_WIRING_TT8 S= tm_err_wiring2.Q;

// NETWORK 13
//   ERR_BURNER_2: AT %MX408.13
ERR_BURNER_2 S= BURNER_2.DA;

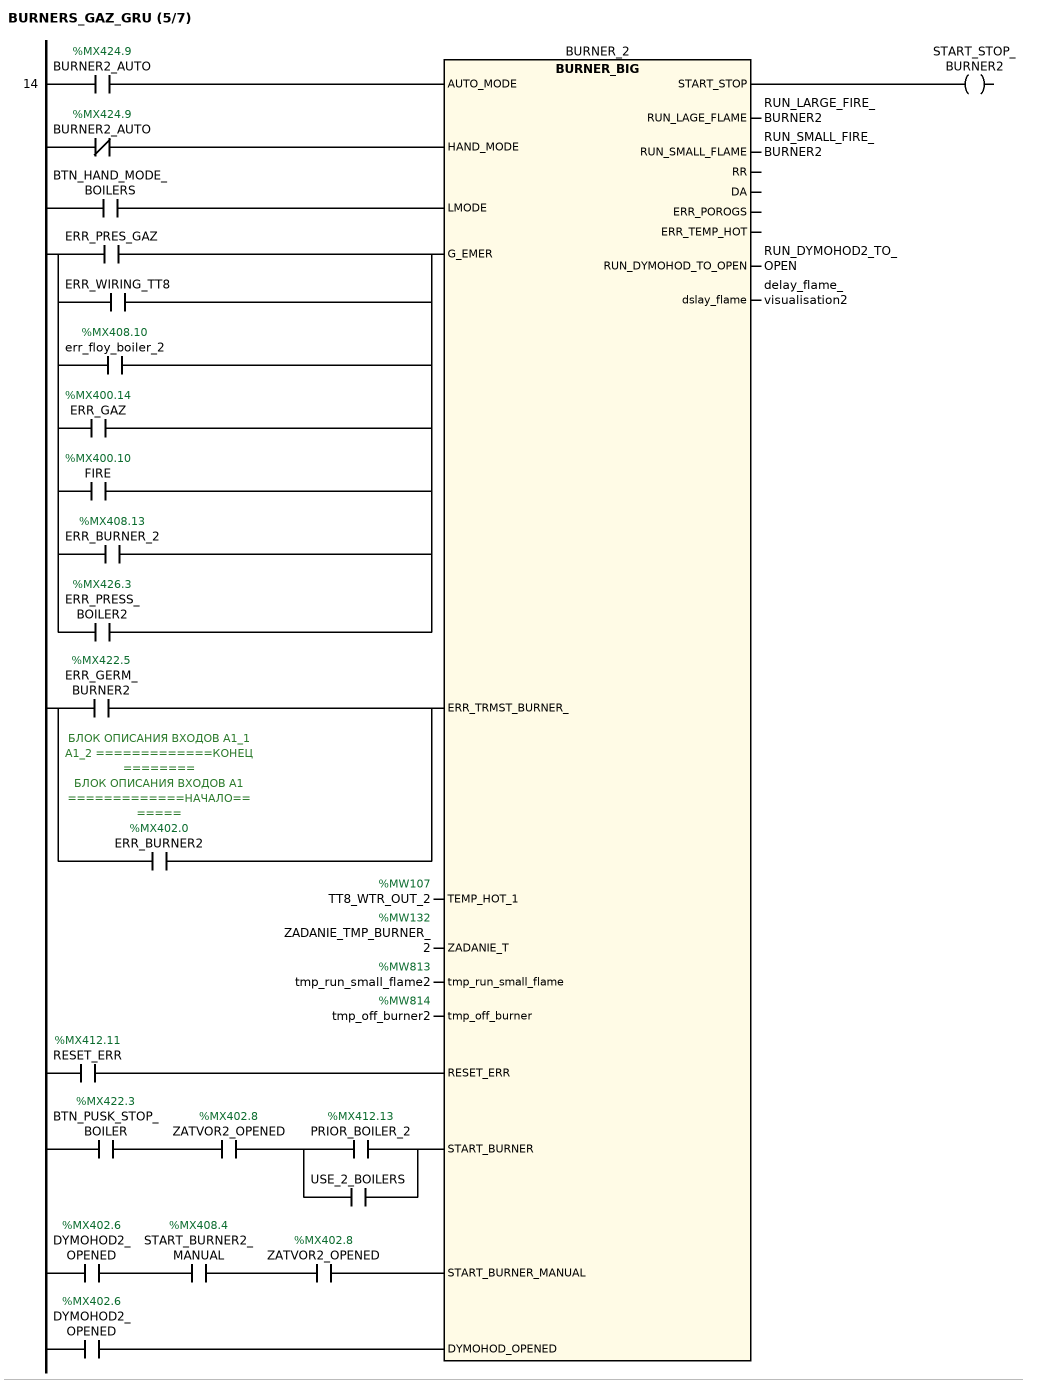
// NETWORK 14
//   BURNER2_AUTO: AT %MX424.9
//   err_floy_boiler_2: AT %MX408.10
//   ERR_GAZ: AT %MX400.14
//   FIRE: AT %MX400.10
//   ERR_BURNER_2: AT %MX408.13
//   ERR_PRESS_BOILER2: AT %MX426.3
//   ERR_GERM_BURNER2: AT %MX422.5
//   ERR_BURNER2: БЛОК ОПИСАНИЯ ВХОДОВ А1_1 A1_2 =============КОНЕЦ======== БЛОК ОПИСАНИЯ ВХОДОВ А1 =============НАЧАЛО======= | AT %MX402.0
//   TT8_WTR_OUT_2: AT %MW107
//   ZADANIE_TMP_BURNER_2: AT %MW132
//   tmp_run_small_flame2: AT %MW813
//   tmp_off_burner2: AT %MW814
//   RESET_ERR: AT %MX412.11
//   BTN_PUSK_STOP_BOILER: AT %MX422.3
//   ZATVOR2_OPENED: AT %MX402.8
//   PRIOR_BOILER_2: AT %MX412.13
//   DYMOHOD2_OPENED: AT %MX402.6
//   START_BURNER2_MANUAL: AT %MX408.4
//   RUN_LARGE_FIRE_BURNER2: AT %MX408.1
//   RUN_SMALL_FIRE_BURNER2: AT %MX408.0
//   delay_flame_visualisation2: AT %MX422.10
BURNER_2(
    AUTO_MODE := BURNER2_AUTO,
    HAND_MODE := NOT BURNER2_AUTO,
    LMODE := BTN_HAND_MODE_BOILERS,
    G_EMER := ERR_PRES_GAZ OR ERR_WIRING_TT8 OR err_floy_boiler_2 OR ERR_GAZ OR FIRE OR ERR_BURNER_2 OR ERR_PRESS_BOILER2,
    ERR_TRMST_BURNER_ := ERR_GERM_BURNER2 OR ERR_BURNER2,
    TEMP_HOT_1 := TT8_WTR_OUT_2,
    ZADANIE_T := ZADANIE_TMP_BURNER_2,
    tmp_run_small_flame := tmp_run_small_flame2,
    tmp_off_burner := tmp_off_burner2,
    RESET_ERR := RESET_ERR,
    START_BURNER := BTN_PUSK_STOP_BOILER AND ZATVOR2_OPENED AND (PRIOR_BOILER_2 OR USE_2_BOILERS),
    START_BURNER_MANUAL := DYMOHOD2_OPENED AND START_BURNER2_MANUAL AND ZATVOR2_OPENED,
    DYMOHOD_OPENED := DYMOHOD2_OPENED,
    RUN_LAGE_FLAME => RUN_LARGE_FIRE_BURNER2,
    RUN_SMALL_FLAME => RUN_SMALL_FIRE_BURNER2,
    RUN_DYMOHOD_TO_OPEN => RUN_DYMOHOD2_TO_OPEN,
    dslay_flame => delay_flame_visualisation2); // BURNER_BIG
START_STOP_BURNER2 := BURNER_2.START_STOP;

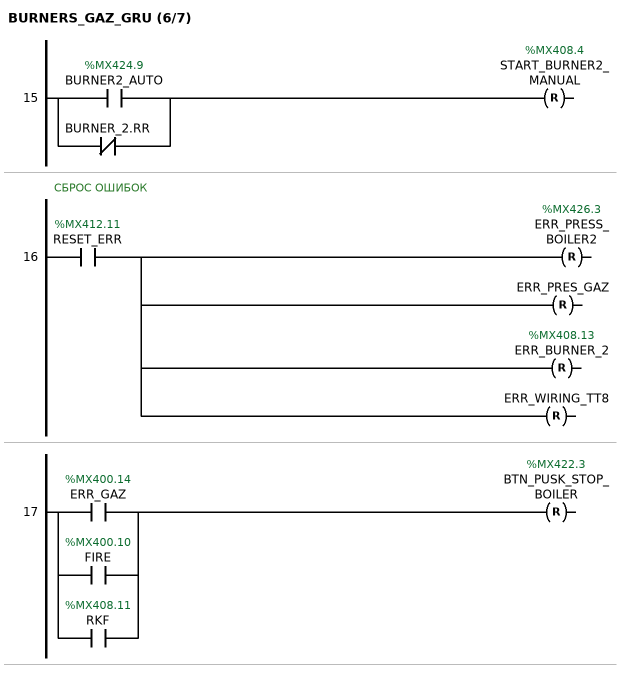
// NETWORK 15
//   BURNER2_AUTO: AT %MX424.9
//   START_BURNER2_MANUAL: AT %MX408.4
START_BURNER2_MANUAL R= BURNER2_AUTO OR NOT BURNER_2.RR;

// NETWORK 16
// СБРОС ОШИБОК
//   RESET_ERR: AT %MX412.11
//   ERR_PRESS_BOILER2: AT %MX426.3
//   ERR_BURNER_2: AT %MX408.13
ERR_PRESS_BOILER2 R= RESET_ERR;
ERR_PRES_GAZ R= RESET_ERR;
ERR_BURNER_2 R= RESET_ERR;
ERR_WIRING_TT8 R= RESET_ERR;

// NETWORK 17
//   ERR_GAZ: AT %MX400.14
//   FIRE: AT %MX400.10
//   RKF: AT %MX408.11
//   BTN_PUSK_STOP_BOILER: AT %MX422.3
BTN_PUSK_STOP_BOILER R= ERR_GAZ OR FIRE OR RKF;

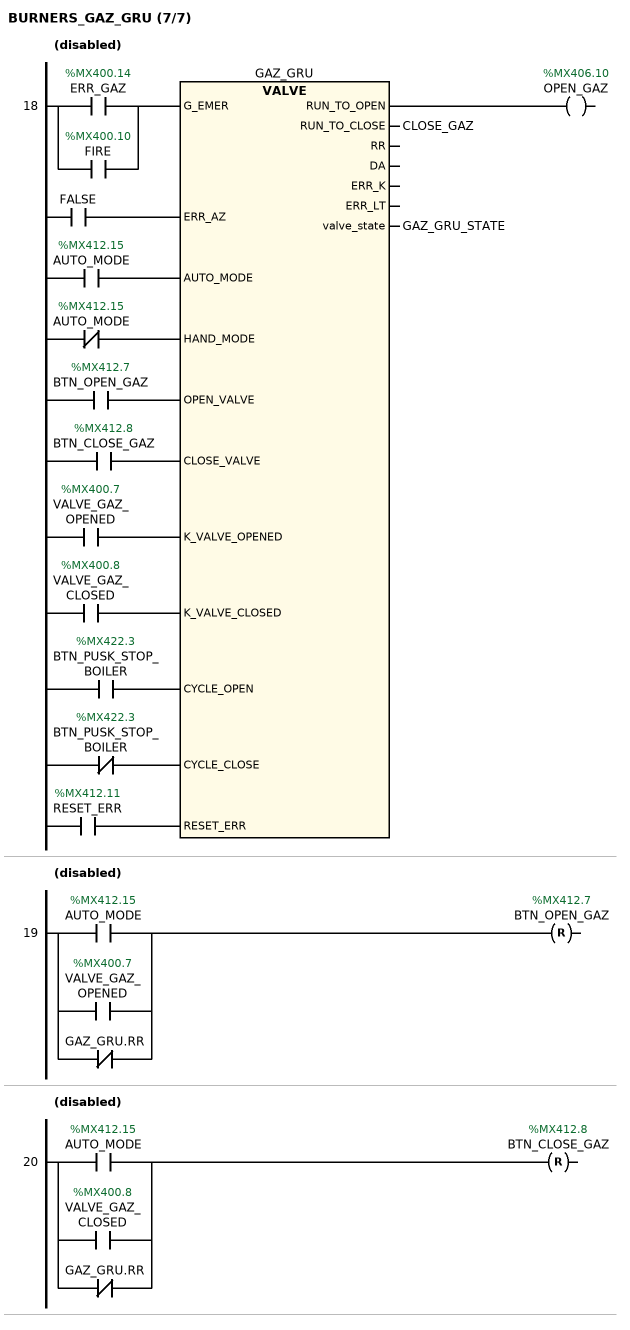
// NETWORK 18 (disabled)
//   ERR_GAZ: AT %MX400.14
//   FIRE: AT %MX400.10
//   AUTO_MODE: AT %MX412.15
//   BTN_OPEN_GAZ: AT %MX412.7
//   BTN_CLOSE_GAZ: AT %MX412.8
//   VALVE_GAZ_OPENED: AT %MX400.7
//   VALVE_GAZ_CLOSED: AT %MX400.8
//   BTN_PUSK_STOP_BOILER: AT %MX422.3
//   RESET_ERR: AT %MX412.11
//   CLOSE_GAZ: AT %MX406.11
//   GAZ_GRU_STATE: AT %MW400
//   OPEN_GAZ: AT %MX406.10
// GAZ_GRU(
//     G_EMER := ERR_GAZ OR FIRE,
//     ERR_AZ := FALSE,
//     AUTO_MODE := AUTO_MODE,
//     HAND_MODE := NOT AUTO_MODE,
//     OPEN_VALVE := BTN_OPEN_GAZ,
//     CLOSE_VALVE := BTN_CLOSE_GAZ,
//     K_VALVE_OPENED := VALVE_GAZ_OPENED,
//     K_VALVE_CLOSED := VALVE_GAZ_CLOSED,
//     CYCLE_OPEN := BTN_PUSK_STOP_BOILER,
//     CYCLE_CLOSE := NOT BTN_PUSK_STOP_BOILER,
//     RESET_ERR := RESET_ERR,
//     RUN_TO_CLOSE => CLOSE_GAZ,
//     valve_state => GAZ_GRU_STATE); // VALVE
// OPEN_GAZ := GAZ_GRU.RUN_TO_OPEN;

// NETWORK 19 (disabled)
//   AUTO_MODE: AT %MX412.15
//   VALVE_GAZ_OPENED: AT %MX400.7
//   BTN_OPEN_GAZ: AT %MX412.7
// BTN_OPEN_GAZ R= AUTO_MODE OR VALVE_GAZ_OPENED OR NOT GAZ_GRU.RR;

// NETWORK 20 (disabled)
//   AUTO_MODE: AT %MX412.15
//   VALVE_GAZ_CLOSED: AT %MX400.8
//   BTN_CLOSE_GAZ: AT %MX412.8
// BTN_CLOSE_GAZ R= AUTO_MODE OR VALVE_GAZ_CLOSED OR NOT GAZ_GRU.RR;

END_PROGRAM

// MyController/Application/FB/BURNER_SMALL
FUNCTION_BLOCK BURNER_SMALL
VAR_INPUT
	AUTO_MODE: BOOL;//АВТОМАТИЧЕСКИ РЕЖИМ
	HAND_MODE: BOOL;//РУЧНОЙ РЕЖИМ
	LMODE: BOOL;//МЕСТНЫЙ РЕЖИМ РАБОТЫ
	G_EMER: BOOL;//АВАРИЙНАЯ ОСТАНОВКА СИСТЕМЫ
	ERR_TRMST_BURNER_: BOOL;//АВАРИЙНЫЙ ТЕРМОСТАТ ГОРЕЛКИ
	TEMP_HOT_1: INT;//ТЕМПЕРАТУРА ГОРЯЧЕГО КАНАЛА 1
	ZADANIE_T: INT;//ПОРОГ ТЕМПЕРАТУРЫ НИЖЕ КОТОРОГО ВКЛЮЧАЕТСЯ 2 СТУПЕНИ
	tmp_run_small_flame: INT;
	tmp_off_burner: INT;
	RESET_ERR: BOOL;
	START_BURNER: BOOL;
	START_BURNER_MANUAL: BOOL;
	DYMOHOD_OPENED: BOOL;
END_VAR
VAR_OUTPUT
	START_STOP: BOOL;//ПУСК/СТОП ГОРЕЛКИ
	RUN_LAGE_FLAME: BOOL;//ВКЛЮЧИТЬ БОЛЬШОЕ ПЛАМЯ
	RUN_SMALL_FLAME: BOOL;//ВКЛЮЧИТЬ МАЛОЕ ПЛАМЯ
	RR: BOOL;
	DA: BOOL;
	ERR_POROGS: BOOL;
	ERR_TEMP_HOT: BOOL;

	RUN_DYMOHOD_TO_OPEN: BOOL;
	
	dslay_flame: BOOL;
END_VAR
VAR
	USE_LAGE_FLAME: BOOL;
	USE_SMALL_FLAME: BOOL;
	ERR_POR_1_2: BOOL;
	ERR_POR_2_3: BOOL;
	ERR_TEMP_HOT_1: BOOL;
	ERR_TEMP_HOT_2: BOOL;
	ERR_TEMP_PROD_3: BOOL;
	TM_UNLOCK_BURNER: TOF;
	tm_err_wiring_t_hot: TON;
	tm_err_temp_hot: TON;
	USE_BURNER: BOOL;
	delay_flame_visualisasion: TON;
END_VAR
VAR // added by the converter: edge detectors and wires of the graphical bodies
    _w1, _w2, _w3, _w4 : BOOL;
END_VAR

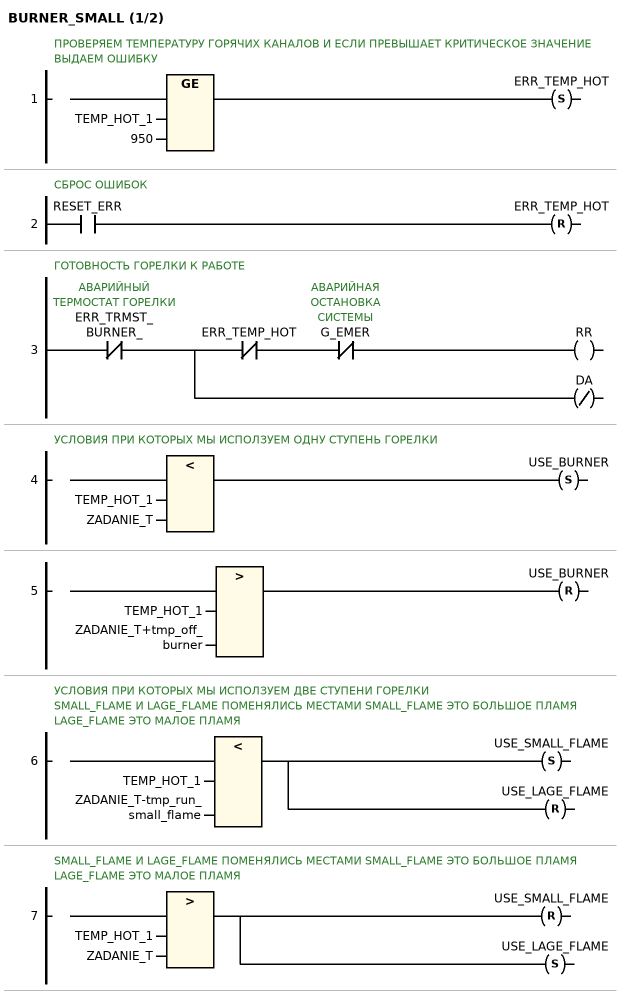
// NETWORK 1
// ПРОВЕРЯЕМ ТЕМПЕРАТУРУ ГОРЯЧИХ КАНАЛОВ И ЕСЛИ ПРЕВЫШАЕТ КРИТИЧЕСКОЕ ЗНАЧЕНИЕ ВЫДАЕМ ОШИБКУ
//   TEMP_HOT_1: ТЕМПЕРАТУРА ГОРЯЧЕГО КАНАЛА 1
ERR_TEMP_HOT S= TEMP_HOT_1 >= 950;

// NETWORK 2
// СБРОС ОШИБОК
ERR_TEMP_HOT R= RESET_ERR;

// NETWORK 3
// ГОТОВНОСТЬ ГОРЕЛКИ К РАБОТЕ
//   ERR_TRMST_BURNER_: АВАРИЙНЫЙ ТЕРМОСТАТ ГОРЕЛКИ
//   G_EMER: АВАРИЙНАЯ ОСТАНОВКА СИСТЕМЫ
_w1 := NOT ERR_TRMST_BURNER_;
RR := _w1 AND NOT ERR_TEMP_HOT AND NOT G_EMER;
DA := NOT _w1;

// NETWORK 4
// УСЛОВИЯ ПРИ КОТОРЫХ МЫ ИСПОЛЗУЕМ ОДНУ СТУПЕНЬ ГОРЕЛКИ
//   TEMP_HOT_1: ТЕМПЕРАТУРА ГОРЯЧЕГО КАНАЛА 1
//   ZADANIE_T: ПОРОГ ТЕМПЕРАТУРЫ НИЖЕ КОТОРОГО ВКЛЮЧАЕТСЯ 2 СТУПЕНИ
USE_BURNER S= TEMP_HOT_1 < ZADANIE_T;

// NETWORK 5
//   TEMP_HOT_1: ТЕМПЕРАТУРА ГОРЯЧЕГО КАНАЛА 1
//   ZADANIE_T+tmp_off_burner: ПОРОГ ТЕМПЕРАТУРЫ НИЖЕ КОТОРОГО ВКЛЮЧАЕТСЯ 2 СТУПЕНИ
USE_BURNER R= TEMP_HOT_1 > (ZADANIE_T+tmp_off_burner);

// NETWORK 6
// УСЛОВИЯ ПРИ КОТОРЫХ МЫ ИСПОЛЗУЕМ ДВЕ СТУПЕНИ ГОРЕЛКИ
// SMALL_FLAME И LAGE_FLAME ПОМЕНЯЛИСЬ МЕСТАМИ SMALL_FLAME ЭТО БОЛЬШОЕ ПЛАМЯ LAGE_FLAME ЭТО МАЛОЕ ПЛАМЯ
//   TEMP_HOT_1: ТЕМПЕРАТУРА ГОРЯЧЕГО КАНАЛА 1
//   ZADANIE_T-tmp_run_small_flame: ПОРОГ ТЕМПЕРАТУРЫ НИЖЕ КОТОРОГО ВКЛЮЧАЕТСЯ 2 СТУПЕНИ
_w2 := TEMP_HOT_1 < (ZADANIE_T-tmp_run_small_flame);
USE_SMALL_FLAME S= _w2;
USE_LAGE_FLAME R= _w2;

// NETWORK 7
// SMALL_FLAME И LAGE_FLAME ПОМЕНЯЛИСЬ МЕСТАМИ SMALL_FLAME ЭТО БОЛЬШОЕ ПЛАМЯ LAGE_FLAME ЭТО МАЛОЕ ПЛАМЯ
//   TEMP_HOT_1: ТЕМПЕРАТУРА ГОРЯЧЕГО КАНАЛА 1
//   ZADANIE_T: ПОРОГ ТЕМПЕРАТУРЫ НИЖЕ КОТОРОГО ВКЛЮЧАЕТСЯ 2 СТУПЕНИ
_w3 := TEMP_HOT_1 > ZADANIE_T;
USE_SMALL_FLAME R= _w3;
USE_LAGE_FLAME S= _w3;

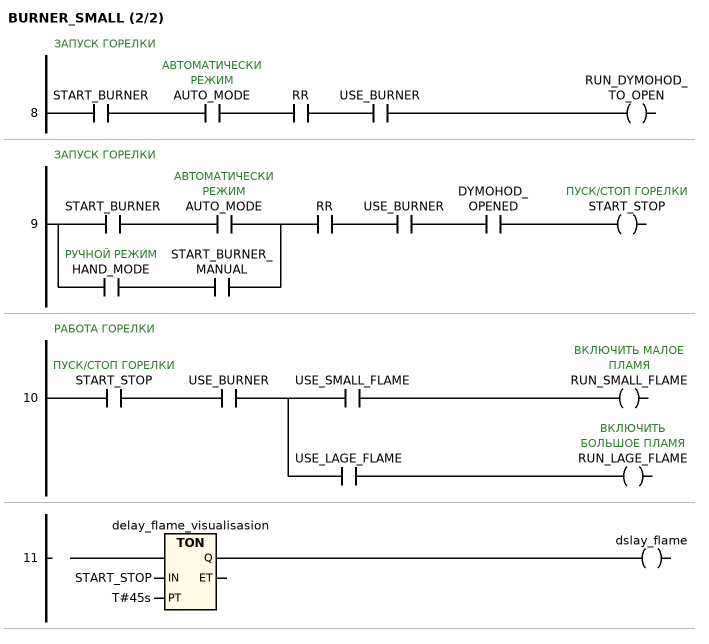
// NETWORK 8
// ЗАПУСК ГОРЕЛКИ
//   AUTO_MODE: АВТОМАТИЧЕСКИ РЕЖИМ
RUN_DYMOHOD_TO_OPEN := START_BURNER AND AUTO_MODE AND RR AND USE_BURNER;

// NETWORK 9
// ЗАПУСК ГОРЕЛКИ
//   AUTO_MODE: АВТОМАТИЧЕСКИ РЕЖИМ
//   HAND_MODE: РУЧНОЙ РЕЖИМ
//   START_STOP: ПУСК/СТОП ГОРЕЛКИ
START_STOP := (START_BURNER AND AUTO_MODE OR HAND_MODE AND START_BURNER_MANUAL) AND RR AND USE_BURNER AND DYMOHOD_OPENED;

// NETWORK 10
// РАБОТА ГОРЕЛКИ
//   START_STOP: ПУСК/СТОП ГОРЕЛКИ
//   RUN_SMALL_FLAME: ВКЛЮЧИТЬ МАЛОЕ ПЛАМЯ
//   RUN_LAGE_FLAME: ВКЛЮЧИТЬ БОЛЬШОЕ ПЛАМЯ
_w4 := START_STOP AND USE_BURNER;
RUN_SMALL_FLAME := _w4 AND USE_SMALL_FLAME;
RUN_LAGE_FLAME := _w4 AND USE_LAGE_FLAME;

// NETWORK 11
//   START_STOP: ПУСК/СТОП ГОРЕЛКИ
delay_flame_visualisasion(IN := START_STOP, PT := T#45s); // TON
dslay_flame := delay_flame_visualisasion.Q;

END_FUNCTION_BLOCK

// MyController/Application/FB/BURNER_BIG
FUNCTION_BLOCK BURNER_BIG
VAR_INPUT
	AUTO_MODE: BOOL;//АВТОМАТИЧЕСКИ РЕЖИМ
	HAND_MODE: BOOL;//РУЧНОЙ РЕЖИМ
	LMODE: BOOL;//МЕСТНЫЙ РЕЖИМ РАБОТЫ
	G_EMER: BOOL;//АВАРИЙНАЯ ОСТАНОВКА СИСТЕМЫ
	ERR_TRMST_BURNER_: BOOL;//АВАРИЙНЫЙ ТЕРМОСТАТ ГОРЕЛКИ
	TEMP_HOT_1: INT;//ТЕМПЕРАТУРА ГОРЯЧЕГО КАНАЛА 1
	ZADANIE_T: INT;//ПОРОГ ТЕМПЕРАТУРЫ НИЖЕ КОТОРОГО ВКЛЮЧАЕТСЯ 2 СТУПЕНИ
	tmp_run_small_flame: INT;
	tmp_off_burner: INT;
	RESET_ERR: BOOL;
	START_BURNER: BOOL;
	START_BURNER_MANUAL: BOOL;
	DYMOHOD_OPENED: BOOL;
END_VAR
VAR_OUTPUT
	START_STOP: BOOL;//ПУСК/СТОП ГОРЕЛКИ
	RUN_LAGE_FLAME: BOOL;//ВКЛЮЧИТЬ БОЛЬШОЕ ПЛАМЯ
	RUN_SMALL_FLAME: BOOL;//ВКЛЮЧИТЬ МАЛОЕ ПЛАМЯ
	RR: BOOL;
	DA: BOOL;
	ERR_POROGS: BOOL;
	ERR_TEMP_HOT: BOOL;

	RUN_DYMOHOD_TO_OPEN: BOOL;
	
	dslay_flame: BOOL;
END_VAR
VAR
	USE_LAGE_FLAME: BOOL;
	USE_SMALL_FLAME: BOOL;
	ERR_POR_1_2: BOOL;
	ERR_POR_2_3: BOOL;
	ERR_TEMP_HOT_1: BOOL;
	ERR_TEMP_HOT_2: BOOL;
	ERR_TEMP_PROD_3: BOOL;
	TM_UNLOCK_BURNER: TOF;
	tm_err_wiring_t_hot: TON;
	tm_err_temp_hot: TON;
	USE_BURNER: BOOL;
	delay_flame_visualisasion: TON;
END_VAR
VAR // added by the converter: edge detectors and wires of the graphical bodies
    _w1, _w2, _w3, _w4 : BOOL;
END_VAR

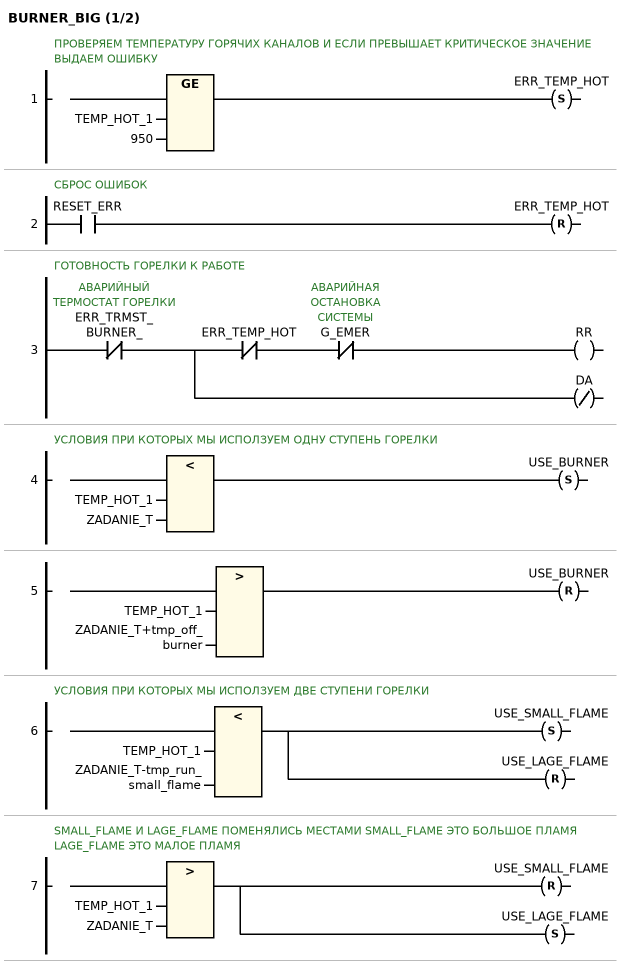
// NETWORK 1
// ПРОВЕРЯЕМ ТЕМПЕРАТУРУ ГОРЯЧИХ КАНАЛОВ И ЕСЛИ ПРЕВЫШАЕТ КРИТИЧЕСКОЕ ЗНАЧЕНИЕ ВЫДАЕМ ОШИБКУ
//   TEMP_HOT_1: ТЕМПЕРАТУРА ГОРЯЧЕГО КАНАЛА 1
ERR_TEMP_HOT S= TEMP_HOT_1 >= 950;

// NETWORK 2
// СБРОС ОШИБОК
ERR_TEMP_HOT R= RESET_ERR;

// NETWORK 3
// ГОТОВНОСТЬ ГОРЕЛКИ К РАБОТЕ
//   ERR_TRMST_BURNER_: АВАРИЙНЫЙ ТЕРМОСТАТ ГОРЕЛКИ
//   G_EMER: АВАРИЙНАЯ ОСТАНОВКА СИСТЕМЫ
_w1 := NOT ERR_TRMST_BURNER_;
RR := _w1 AND NOT ERR_TEMP_HOT AND NOT G_EMER;
DA := NOT _w1;

// NETWORK 4
// УСЛОВИЯ ПРИ КОТОРЫХ МЫ ИСПОЛЗУЕМ ОДНУ СТУПЕНЬ ГОРЕЛКИ
//   TEMP_HOT_1: ТЕМПЕРАТУРА ГОРЯЧЕГО КАНАЛА 1
//   ZADANIE_T: ПОРОГ ТЕМПЕРАТУРЫ НИЖЕ КОТОРОГО ВКЛЮЧАЕТСЯ 2 СТУПЕНИ
USE_BURNER S= TEMP_HOT_1 < ZADANIE_T;

// NETWORK 5
//   TEMP_HOT_1: ТЕМПЕРАТУРА ГОРЯЧЕГО КАНАЛА 1
//   ZADANIE_T+tmp_off_burner: ПОРОГ ТЕМПЕРАТУРЫ НИЖЕ КОТОРОГО ВКЛЮЧАЕТСЯ 2 СТУПЕНИ
USE_BURNER R= TEMP_HOT_1 > (ZADANIE_T+tmp_off_burner);

// NETWORK 6
// УСЛОВИЯ ПРИ КОТОРЫХ МЫ ИСПОЛЗУЕМ ДВЕ СТУПЕНИ ГОРЕЛКИ
//   TEMP_HOT_1: ТЕМПЕРАТУРА ГОРЯЧЕГО КАНАЛА 1
//   ZADANIE_T-tmp_run_small_flame: ПОРОГ ТЕМПЕРАТУРЫ НИЖЕ КОТОРОГО ВКЛЮЧАЕТСЯ 2 СТУПЕНИ
_w2 := TEMP_HOT_1 < (ZADANIE_T-tmp_run_small_flame);
USE_SMALL_FLAME S= _w2;
USE_LAGE_FLAME R= _w2;

// NETWORK 7
// SMALL_FLAME И LAGE_FLAME ПОМЕНЯЛИСЬ МЕСТАМИ SMALL_FLAME ЭТО БОЛЬШОЕ ПЛАМЯ LAGE_FLAME ЭТО МАЛОЕ ПЛАМЯ
//   TEMP_HOT_1: ТЕМПЕРАТУРА ГОРЯЧЕГО КАНАЛА 1
//   ZADANIE_T: ПОРОГ ТЕМПЕРАТУРЫ НИЖЕ КОТОРОГО ВКЛЮЧАЕТСЯ 2 СТУПЕНИ
_w3 := TEMP_HOT_1 > ZADANIE_T;
USE_SMALL_FLAME R= _w3;
USE_LAGE_FLAME S= _w3;

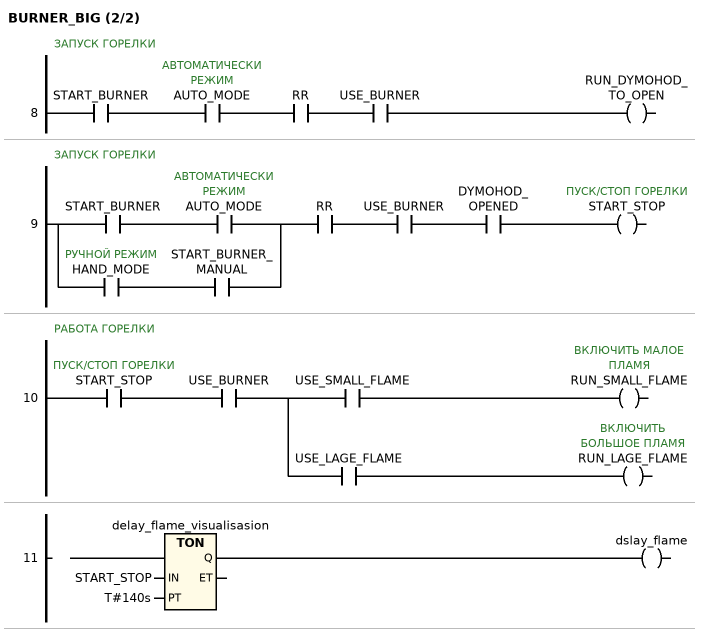
// NETWORK 8
// ЗАПУСК ГОРЕЛКИ
//   AUTO_MODE: АВТОМАТИЧЕСКИ РЕЖИМ
RUN_DYMOHOD_TO_OPEN := START_BURNER AND AUTO_MODE AND RR AND USE_BURNER;

// NETWORK 9
// ЗАПУСК ГОРЕЛКИ
//   AUTO_MODE: АВТОМАТИЧЕСКИ РЕЖИМ
//   HAND_MODE: РУЧНОЙ РЕЖИМ
//   START_STOP: ПУСК/СТОП ГОРЕЛКИ
START_STOP := (START_BURNER AND AUTO_MODE OR HAND_MODE AND START_BURNER_MANUAL) AND RR AND USE_BURNER AND DYMOHOD_OPENED;

// NETWORK 10
// РАБОТА ГОРЕЛКИ
//   START_STOP: ПУСК/СТОП ГОРЕЛКИ
//   RUN_SMALL_FLAME: ВКЛЮЧИТЬ МАЛОЕ ПЛАМЯ
//   RUN_LAGE_FLAME: ВКЛЮЧИТЬ БОЛЬШОЕ ПЛАМЯ
_w4 := START_STOP AND USE_BURNER;
RUN_SMALL_FLAME := _w4 AND USE_SMALL_FLAME;
RUN_LAGE_FLAME := _w4 AND USE_LAGE_FLAME;

// NETWORK 11
//   START_STOP: ПУСК/СТОП ГОРЕЛКИ
delay_flame_visualisasion(IN := START_STOP, PT := T#140s); // TON
dslay_flame := delay_flame_visualisasion.Q;

END_FUNCTION_BLOCK

// MyController/Application/FB/VALVE
FUNCTION_BLOCK VALVE
VAR_INPUT
	G_EMER: BOOL;
	ERR_AZ: BOOL;
	AUTO_MODE: BOOL;
	HAND_MODE: BOOL;
	OPEN_VALVE: BOOL;
	CLOSE_VALVE: BOOL;
	K_VALVE_OPENED: BOOL;
	K_VALVE_CLOSED: BOOL;
	CYCLE_OPEN: BOOL;
	CYCLE_CLOSE: BOOL;
	RESET_ERR: BOOL;	
END_VAR
VAR_OUTPUT
	RUN_TO_OPEN: BOOL;
	RUN_TO_CLOSE: BOOL;
	RR: BOOL;
	DA: BOOL;
	ERR_K: BOOL;
	ERR_LT: BOOL;
	valve_state: BYTE;
END_VAR
VAR
	TM_LT_VALVE: TON;
END_VAR
VAR // added by the converter: edge detectors and wires of the graphical bodies
    _w1 : BOOL;
END_VAR

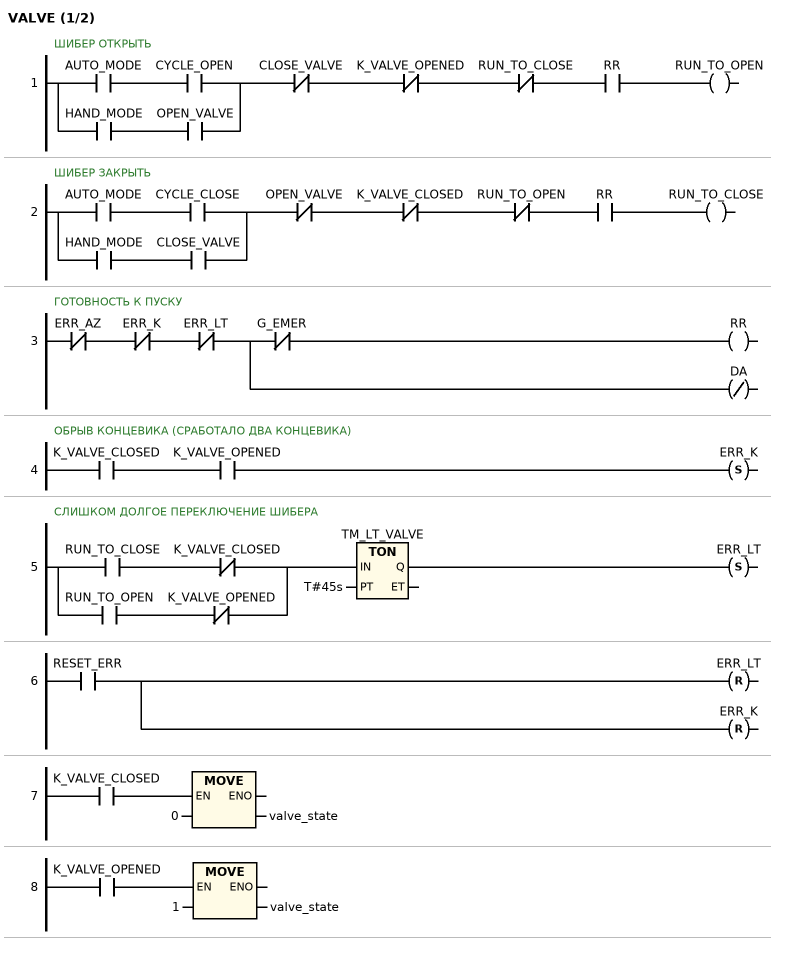
// NETWORK 1
// ШИБЕР ОТКРЫТЬ
RUN_TO_OPEN := (AUTO_MODE AND CYCLE_OPEN OR HAND_MODE AND OPEN_VALVE) AND NOT CLOSE_VALVE AND NOT K_VALVE_OPENED AND NOT RUN_TO_CLOSE AND RR;

// NETWORK 2
// ШИБЕР ЗАКРЫТЬ
RUN_TO_CLOSE := (AUTO_MODE AND CYCLE_CLOSE OR HAND_MODE AND CLOSE_VALVE) AND NOT OPEN_VALVE AND NOT K_VALVE_CLOSED AND NOT RUN_TO_OPEN AND RR;

// NETWORK 3
// ГОТОВНОСТЬ К ПУСКУ
_w1 := NOT ERR_AZ AND NOT ERR_K AND NOT ERR_LT;
RR := _w1 AND NOT G_EMER;
DA := NOT _w1;

// NETWORK 4
// ОБРЫВ КОНЦЕВИКА (СРАБОТАЛО ДВА КОНЦЕВИКА)
ERR_K S= K_VALVE_CLOSED AND K_VALVE_OPENED;

// NETWORK 5
// СЛИШКОМ ДОЛГОЕ ПЕРЕКЛЮЧЕНИЕ ШИБЕРА
TM_LT_VALVE(IN := RUN_TO_CLOSE AND NOT K_VALVE_CLOSED OR RUN_TO_OPEN AND NOT K_VALVE_OPENED, PT := T#45s); // TON
ERR_LT S= TM_LT_VALVE.Q;

// NETWORK 6
ERR_LT R= RESET_ERR;
ERR_K R= RESET_ERR;

// NETWORK 7
IF K_VALVE_CLOSED THEN valve_state := 0; END_IF

// NETWORK 8
IF K_VALVE_OPENED THEN valve_state := 1; END_IF

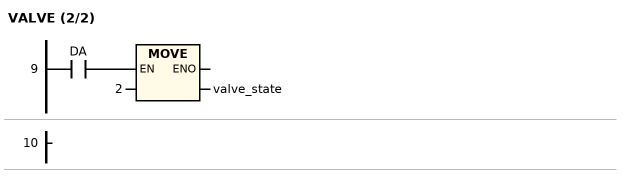
// NETWORK 9
IF DA THEN valve_state := 2; END_IF

// NETWORK 10

END_FUNCTION_BLOCK

// MyController/Application/avg
PROGRAM avg
VAR
	avg_balanse: STATISTICS_INT;
	utilizator: INTEGRAL;
	power_utilizator_za_min: REAL;
END_VAR

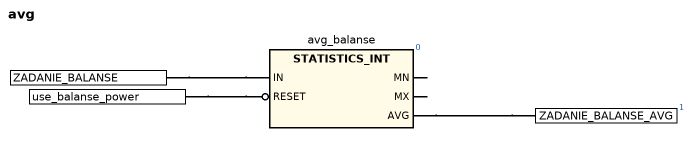
avg_balanse(IN := ZADANIE_BALANSE, RESET := NOT use_balanse_power); // STATISTICS_INT
ZADANIE_BALANSE_AVG := avg_balanse.AVG;

END_PROGRAM

// MyController/Application/day_mode
PROGRAM day_mode
VAR
      uidResultRtcGet: UDINT;
      stGetDate: SysTimeRtc.RTS_SYSTIMEDATE; 
      uiGetYear: UINT; 
      uiGetMonth: UINT; 
      uiGetDay: UINT; 
      uiGetHour: UINT; 
      uiGetMinute: UINT; 
      uiGetSecond: UINT; 
      uiGetMSecond: UINT; 
      uiGetDayOfWeek: UINT; 
      uiGetYday: UINT; 
      uidResultConvertToDate: UDINT; 

END_VAR
VAR // added by the converter: edge detectors and wires of the graphical bodies
    _w1 : ANY;
    _w2 : BOOL;
END_VAR

_w1 := SysTimeRtcGet(pResult := uidResultRtcGet);
IF _w2 THEN SysTimeRtcConvertUtcToDate(dwTimestampUtc := _w1, pDate := stGetDate); END_IF
_w2 := uidResultRtcGet = 16#0;
uiGetYear := stGetDate.RTS_SYSTIMEDATE;
uiGetMonth := stGetDate.wYear;
uiGetDay := stGetDate.wMonth;
uiGetHour := stGetDate.wDay;
uiGetMinute := stGetDate.wHour;
uiGetSecond := stGetDate.wMinute;
uiGetMSecond := stGetDate.wSecond;
uiGetDayOfWeek := stGetDate.wMilliseconds;
uiGetYday := stGetDate.wDayOfWeek;

END_PROGRAM

// MyController/Application/HVO_HEATER
PROGRAM HVO_HEATER
VAR
	HV: BYTE;
	
	PID_HEATER: PID;
	cycle_hvo_run_open: BOOL;
	cycle_hvo_run_close: BOOL;
END_VAR
VAR // added by the converter: edge detectors and wires of the graphical bodies
    _w1, _w2 : BOOL;
    _rt1, _rt2 : R_TRIG;
END_VAR

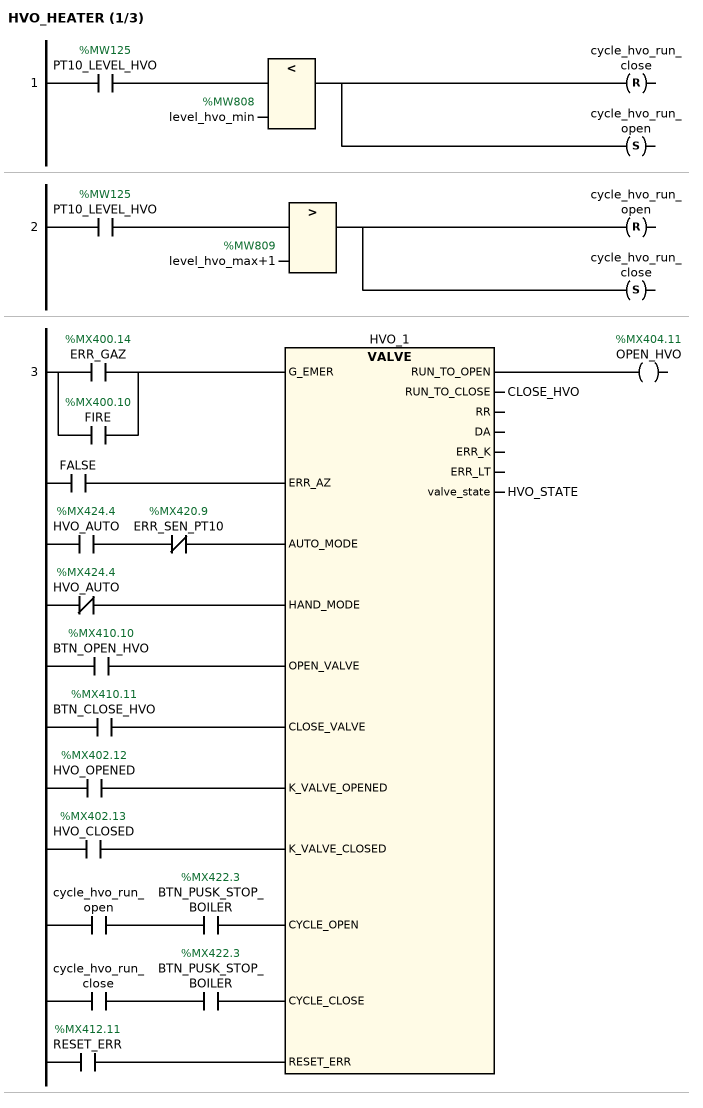
// NETWORK 1
//   PT10_LEVEL_HVO: AT %MW125
//   level_hvo_min: AT %MW808
_w1 := PT10_LEVEL_HVO < level_hvo_min;
cycle_hvo_run_close R= _w1;
cycle_hvo_run_open S= _w1;

// NETWORK 2
//   PT10_LEVEL_HVO: AT %MW125
//   level_hvo_max+1: AT %MW809
_w2 := PT10_LEVEL_HVO > (level_hvo_max+1);
cycle_hvo_run_open R= _w2;
cycle_hvo_run_close S= _w2;

// NETWORK 3
//   ERR_GAZ: AT %MX400.14
//   FIRE: AT %MX400.10
//   HVO_AUTO: AT %MX424.4
//   ERR_SEN_PT10: AT %MX420.9
//   BTN_OPEN_HVO: AT %MX410.10
//   BTN_CLOSE_HVO: AT %MX410.11
//   HVO_OPENED: AT %MX402.12
//   HVO_CLOSED: AT %MX402.13
//   BTN_PUSK_STOP_BOILER: AT %MX422.3
//   RESET_ERR: AT %MX412.11
//   CLOSE_HVO: AT %MX404.12
//   HVO_STATE: AT %MW403
//   OPEN_HVO: AT %MX404.11
HVO_1(
    G_EMER := ERR_GAZ OR FIRE,
    ERR_AZ := FALSE,
    AUTO_MODE := HVO_AUTO AND NOT ERR_SEN_PT10,
    HAND_MODE := NOT HVO_AUTO,
    OPEN_VALVE := BTN_OPEN_HVO,
    CLOSE_VALVE := BTN_CLOSE_HVO,
    K_VALVE_OPENED := HVO_OPENED,
    K_VALVE_CLOSED := HVO_CLOSED,
    CYCLE_OPEN := cycle_hvo_run_open AND BTN_PUSK_STOP_BOILER,
    CYCLE_CLOSE := cycle_hvo_run_close AND BTN_PUSK_STOP_BOILER,
    RESET_ERR := RESET_ERR,
    RUN_TO_CLOSE => CLOSE_HVO,
    valve_state => HVO_STATE); // VALVE
OPEN_HVO := HVO_1.RUN_TO_OPEN;

